# B&R Automation Studio project TD52 (part 72)

#### rtwtypes.h
```c
/********************************************************************
 * COPYRIGHT -- Bernecker + Rainer Industrie-Elektronik Ges.m.b.H.
 ********************************************************************
 * Program: LamStart
 * File: rtwtypes.h
 * Author: 105055527
 * Created: Thu May 18 17:26:11 2017
 ********************************************************************
 * Header for program LamStart
 ********************************************************************
 * Generated with B&R Automation Studio Target for Simulink V4.2
 * (ERT based)
 ********************************************************************/

#ifndef __RTWTYPES_H__
#define __RTWTYPES_H__
#ifndef TRUE
# define TRUE                          (1U)
#endif

#ifndef FALSE
# define FALSE                         (0U)
#endif

#ifndef __TMWTYPES__
#define __TMWTYPES__
#include <limits.h>

/*=======================================================================*
 * Target hardware information
 *   Device type: Intel->x86/Pentium
 *   Number of bits:     char:   8    short:   16    long:  32
 *                       long:  32
 *                       native word size:  32
 *   Byte ordering: LittleEndian
 *   Signed integer division rounds to: Zero
 *   Shift right on a signed integer as arithmetic shift: on
 *=======================================================================*/

/*=======================================================================*
 * Fixed width word size data types:                                     *
 *   int8_T, int16_T, int32_T     - signed 8, 16, or 32 bit integers     *
 *   uint8_T, uint16_T, uint32_T  - unsigned 8, 16, or 32 bit integers   *
 *   real32_T, real64_T           - 32 and 64 bit floating point numbers *
 *=======================================================================*/
typedef signed char int8_T;
typedef unsigned char uint8_T;
typedef short int16_T;
typedef unsigned short uint16_T;
typedef long int32_T;
typedef unsigned long uint32_T;
typedef float real32_T;
typedef double real64_T;

/*===========================================================================*
 * Generic type definitions: real_T, time_T, boolean_T, int_T, uint_T,       *
 *                           ulong_T, char_T and byte_T.                     *
 *===========================================================================*/
typedef double real_T;
typedef double time_T;
typedef unsigned char boolean_T;
typedef long int_T;
typedef unsigned long uint_T;
typedef unsigned long ulong_T;
typedef char char_T;
typedef unsigned char uchar_T;
typedef char_T byte_T;

/*=======================================================================*
 * Min and Max:                                                          *
 *   int8_T, int16_T, int32_T     - signed 8, 16, or 32 bit integers     *
 *   uint8_T, uint16_T, uint32_T  - unsigned 8, 16, or 32 bit integers   *
 *=======================================================================*/
#define MAX_int8_T                     ((int8_T)(127))
#define MIN_int8_T                     ((int8_T)(-128))
#define MAX_uint8_T                    ((uint8_T)(255U))
#define MIN_uint8_T                    ((uint8_T)(0U))
#define MAX_int16_T                    ((int16_T)(32767))
#define MIN_int16_T                    ((int16_T)(-32768))
#define MAX_uint16_T                   ((uint16_T)(65535U))
#define MIN_uint16_T                   ((uint16_T)(0U))
#define MAX_int32_T                    ((int32_T)(2147483647))
#define MIN_int32_T                    ((int32_T)(-2147483647-1))
#define MAX_uint32_T                   ((uint32_T)(0xFFFFFFFFU))
#define MIN_uint32_T                   ((uint32_T)(0U))

/* Logical type definitions */
#if (!defined(__cplusplus)) && (!defined(__true_false_are_keywords))
#  ifndef false
#   define false                       (0U)
#  endif

#  ifndef true
#   define true                        (1U)
#  endif
#endif

/*
 * Simulink Coder assumes the code is compiled on a target using a 2's complement representation
 * for signed integer values.
 */
#if ((SCHAR_MIN + 1) != -SCHAR_MAX)
#error "This code must be compiled using a 2's complement representation for signed integer values"
#endif

/* This ID is used to detect inclusion of an incompatible rtwtypes.h */
#define RTWTYPES_ID_C08S16I32L32N32F1
#else                                  /* __TMWTYPES__ */
#define TMWTYPES_PREVIOUSLY_INCLUDED
#endif                                 /* __TMWTYPES__ */

/* Block D-Work pointer type */
typedef void * pointer_T;

/* Simulink specific types */
#ifndef __SIMSTRUC_TYPES_H__
#define __SIMSTRUC_TYPES_H__

/* Trigger directions: falling, either, and rising */
typedef enum {
  FALLING_ZERO_CROSSING = -1,
  ANY_ZERO_CROSSING = 0,
  RISING_ZERO_CROSSING = 1
} ZCDirection;

/* Previous state of a trigger signal */
typedef uint8_T ZCSigState;

/* Initial value of a trigger zero crossing signal */
#define UNINITIALIZED_ZCSIG            0x03U
#define NEG_ZCSIG                      0x02U
#define POS_ZCSIG                      0x01U
#define ZERO_ZCSIG                     0x00U

/* Current state of a trigger signal */
typedef enum {
  FALLING_ZCEVENT = -1,
  NO_ZCEVENT = 0,
  RISING_ZCEVENT = 1
} ZCEventType;

#endif                                 /* __SIMSTRUC_TYPES_H__ */
#endif                                 /* __RTWTYPES_H__ */

#ifndef MIN
#define MIN(a,b)                       ((a) < (b) ? (a) : (b))
#endif

#ifndef MAX
#define MAX(a,b)                       ((a) > (b) ? (a) : (b))
#endif
```

#### LamStart.c
```c
/********************************************************************
 * COPYRIGHT -- Bernecker + Rainer Industrie-Elektronik Ges.m.b.H.
 ********************************************************************
 * Program: LamStart
 * File: LamStart.c
 * Author: 105055527
 * Created: Thu May 18 17:26:11 2017
 ********************************************************************
 * Implementation of program LamStart
 ********************************************************************
 * Generated with B&R Automation Studio Target for Simulink V4.2
 * (ERT based)
 ********************************************************************/
#include "LamStart.h"
#include "LamStart_private.h"

/*  Defines */
#define LamStart_POS_ZCSIG             ((uint8_T)1U)
#define LamStart_UNINITIALIZED_ZCSIG   ((uint8_T)3U)

/*  Data Types */

/**************************** GLOBAL DATA *************************************/
/*  Definitions */

/*  Declarations  */

/***************************** FILE SCOPE DATA ********************************/

/*************************** FUNCTIONS ****************************************/

/* Lookup Binary Search Utility BINARYSEARCH_real32_T */
void BINARYSEARCH_real32_T(uint32_T *piLeft, uint32_T *piRght, real32_T u, const
  real32_T *pData, uint32_T iHi, struct fLamStart* inst)
{
  /* Find the location of current input value in the data table. */
  *piLeft = 0U;
  *piRght = iHi;
  if (u <= pData[0] ) {
    /* Less than or equal to the smallest point in the table. */
    *piRght = 0U;
  } else if (u >= pData[iHi] ) {
    /* Greater than or equal to the largest point in the table. */
    *piLeft = iHi;
  } else {
    uint32_T i;

    /* Do a binary search. */
    while (( *piRght - *piLeft ) > 1U ) {
      /* Get the average of the left and right indices using to Floor rounding. */
      i = (*piLeft + *piRght) >> 1;

      /* Move either the right index or the left index so that */
      /*  LeftDataPoint <= CurrentValue < RightDataPoint */
      if (u < pData[i] ) {
        *piRght = i;
      } else {
        *piLeft = i;
      }
    }
  }
}

/* Lookup Utility LookUp_real32_T_real32_T */
void LookUp_real32_T_real32_T(real32_T *pY, const real32_T *pYData, real32_T u,
  const real32_T *pUData, uint32_T iHi, struct fLamStart* inst)
{
  uint32_T iLeft;
  uint32_T iRght;
  BINARYSEARCH_real32_T( &(iLeft), &(iRght), u, pUData, iHi, inst);

  {
    real32_T lambda;
    if (pUData[iRght] > pUData[iLeft] ) {
      real32_T num;
      real32_T den;
      den = pUData[iRght];
      den = den - pUData[iLeft];
      num = u;
      num = num - pUData[iLeft];
      lambda = num / den;
    } else {
      lambda = 0.0F;
    }

    {
      real32_T yLeftCast;
      real32_T yRghtCast;
      yLeftCast = pYData[iLeft];
      yRghtCast = pYData[iRght];
      yLeftCast += lambda * ( yRghtCast - yLeftCast );
      (*pY) = yLeftCast;
    }
  }
}

/* Model step function */
void LamStart_step(struct BlockIO_LamStart *LamStart_B, struct D_Work_LamStart *LamStart_DWork,
                   struct PrevZCSigStates_LamStart *LamStart_PrevZCSigState,
                   ExternalOutputs_LamStart *LamStart_Y, struct fLamStart* inst)
{
  /* local block i/o variables */
  real32_T rtb_LookupTableDynamic;
  real32_T rtb_TmpSignalConversionAtLookup[2];
  real32_T rtb_TmpSignalConversionAtLook_b[2];
  real32_T rtb_rLowerOilTemp;
  real32_T rtb_rLamLoLim_N_y[3];
  real32_T rtb_rLamLoLim_N_x[3];
  real32_T rtb_rN_Eng_h;
  real32_T rtb_LookupTableDynamic1;
  real32_T rtb_rT_EO;
  boolean_T rtb_LogicalOperator2;
  boolean_T didZcEventOccur;
  real32_T rtb_rHigherOilTemp;
  real32_T rtb_Abs1;
  real32_T rtb_Product;
  real32_T rtb_UkYk1;
  boolean_T rtb_Switch1;
  boolean_T rtb_RelationalOperator;

  /* S-Function (bur_bus_in): '<Root>/Bus Input2' */
  LamStart_B->BusInput2 = inst->Perm;

  /* Abs: '<S6>/Abs1' incorporates:
   *  BusSelector: '<S6>/Bus Selector7'
   */
  rtb_Abs1 = (real32_T)fabs(LamStart_B->BusInput2.rLamSlewRate);

  /* Product: '<S9>/delta rise limit' incorporates:
   *  SampleTimeMath: '<S9>/sample time'
   *
   * About '<S9>/sample time':
   *  y = K where K = ( w * Ts )
   */
  rtb_rHigherOilTemp = rtb_Abs1 * 0.01F;

  /* S-Function (bur_bus_in): '<Root>/Bus Input1' */
  LamStart_B->BusInput1 = inst->Para;

  /* S-Function (bur_bus_in): '<Root>/Bus Input' */
  LamStart_B->BusInput = inst->IN;

  /* BusSelector: '<Root>/Bus Selector3' */
  rtb_rLowerOilTemp = LamStart_B->BusInput.rN_Eng;

  /* BusSelector: '<Root>/Bus Selector13' */
  rtb_rLamLoLim_N_y[0] = LamStart_B->BusInput2.refPoint_Lam_N_Offs_x[0];
  rtb_rLamLoLim_N_y[1] = LamStart_B->BusInput2.refPoint_Lam_N_Offs_x[1];
  rtb_rLamLoLim_N_y[2] = LamStart_B->BusInput2.refPoint_Lam_N_Offs_x[2];
  rtb_rLamLoLim_N_x[0] = LamStart_B->BusInput2.refPoint_Lam_N_Offs_y[0];
  rtb_rLamLoLim_N_x[1] = LamStart_B->BusInput2.refPoint_Lam_N_Offs_y[1];
  rtb_rLamLoLim_N_x[2] = LamStart_B->BusInput2.refPoint_Lam_N_Offs_y[2];

  /* Dynamic Look-Up Table Block: '<Root>/Lookup Table Dynamic2'
   * Input0  Data Type:  Floating Point real32_T
   * Input1  Data Type:  Floating Point real32_T
   * Input2  Data Type:  Floating Point real32_T
   * Output0 Data Type:  Floating Point real32_T
   * Lookup Method: Linear_Endpoint
   *
   */
  LookUp_real32_T_real32_T( &(rtb_rT_EO), rtb_rLamLoLim_N_x, rtb_rLowerOilTemp,
    rtb_rLamLoLim_N_y, 2U, inst);

  /* Product: '<Root>/Product' */
  rtb_Product = LamStart_B->BusInput1.rLam_Start_Offs * rtb_rT_EO;

  /* Switch: '<S7>/Switch3' incorporates:
   *  Constant: '<S6>/Constant2'
   *  Constant: '<S6>/Constant4'
   *  Gain: '<S6>/Gain1'
   *  RelationalOperator: '<S7>/groesser '
   *  RelationalOperator: '<S7>/kleiner'
   *  Switch: '<S7>/Switch1'
   *  Switch: '<S7>/Switch2'
   *  UnitDelay: '<S7>/Unit Delay2'
   */
  if (LamStart_B->BusInput.bReset) {
    rtb_Switch1 = FALSE;
  } else if (LamStart_B->BusInput.rN_Eng < 10.0F) {
    /* Switch: '<S7>/Switch1' incorporates:
     *  Constant: '<S7>/FALSE'
     */
    rtb_Switch1 = FALSE;
  } else if (LamStart_B->BusInput.rN_Eng > 0.995F *
             LamStart_B->BusInput1.rN_EngNom) {
    /* Switch: '<S7>/Switch2' incorporates:
     *  Constant: '<S7>/TRUE'
     *  Switch: '<S7>/Switch1'
     */
    rtb_Switch1 = TRUE;
  } else {
    rtb_Switch1 = LamStart_DWork->UnitDelay2_DSTATE;
  }

  /* End of Switch: '<S7>/Switch3' */

  /* Outputs for Atomic SubSystem: '<S6>/TON' */
  /* Logic: '<S8>/Logical Operator2' */
  rtb_LogicalOperator2 = !rtb_Switch1;

  /* DiscreteIntegrator: '<S8>/Discrete-Time Integrator' */
  if (rtb_LogicalOperator2 || (LamStart_DWork->DiscreteTimeIntegrator_PrevRese
       != 0)) {
    LamStart_DWork->DiscreteTimeIntegrator_DSTATE = 0.0F;
  }

  /* RelationalOperator: '<S8>/Relational Operator' incorporates:
   *  DiscreteIntegrator: '<S8>/Discrete-Time Integrator'
   */
  rtb_RelationalOperator = (LamStart_DWork->DiscreteTimeIntegrator_DSTATE >=
    LamStart_B->BusInput2.rTi_idle);

  /* Update for DiscreteIntegrator: '<S8>/Discrete-Time Integrator' incorporates:
   *  DataTypeConversion: '<S10>/Conversion'
   *  Logic: '<S8>/Logical Operator'
   *  Logic: '<S8>/Logical Operator1'
   */
  LamStart_DWork->DiscreteTimeIntegrator_DSTATE += (real32_T)
    ((!rtb_RelationalOperator) && rtb_Switch1) * 0.01F;
  if (rtb_LogicalOperator2) {
    LamStart_DWork->DiscreteTimeIntegrator_PrevRese = 1;
  } else {
    LamStart_DWork->DiscreteTimeIntegrator_PrevRese = 0;
  }

  /* End of Update for DiscreteIntegrator: '<S8>/Discrete-Time Integrator' */

  /* Logic: '<S6>/Logical Operator' incorporates:
   *  Logic: '<S6>/Logical Operator1'
   *  Logic: '<S8>/Logical Operator3'
   */
  rtb_RelationalOperator = !((rtb_RelationalOperator && rtb_Switch1) ||
    LamStart_B->BusInput.bGCB_ON);

  /* End of Outputs for SubSystem: '<S6>/TON' */

  /* Delay: '<S9>/Delay' */
  didZcEventOccur = (((LamStart_PrevZCSigState->Delay_Reset_ZCE ==
                       LamStart_POS_ZCSIG) != rtb_RelationalOperator) &&
                     (LamStart_PrevZCSigState->Delay_Reset_ZCE !=
                      LamStart_UNINITIALIZED_ZCSIG));
  LamStart_PrevZCSigState->Delay_Reset_ZCE = (uint8_T)rtb_RelationalOperator;
  if (rtb_RelationalOperator || didZcEventOccur) {
    LamStart_DWork->icLoad = 1U;
  }

  if (LamStart_DWork->icLoad != 0) {
    LamStart_DWork->Delay_DSTATE = rtb_Product;
  }

  rtb_rT_EO = LamStart_DWork->Delay_DSTATE;

  /* End of Delay: '<S9>/Delay' */

  /* Switch: '<S9>/etaVolConst' incorporates:
   *  Constant: '<S6>/Constant6'
   */
  if (rtb_RelationalOperator) {
    rtb_UkYk1 = rtb_Product;
  } else {
    rtb_UkYk1 = 0.0F;
  }

  /* End of Switch: '<S9>/etaVolConst' */

  /* Sum: '<S9>/Difference Inputs1' */
  rtb_UkYk1 -= rtb_rT_EO;

  /* Switch: '<S11>/Switch2' incorporates:
   *  RelationalOperator: '<S11>/LowerRelop1'
   */
  if (!(rtb_UkYk1 > rtb_rHigherOilTemp)) {
    /* Product: '<S9>/delta fall limit' incorporates:
     *  Gain: '<S6>/Gain'
     */
    rtb_Abs1 = -rtb_Abs1 * 0.01F;

    /* Switch: '<S11>/Switch' incorporates:
     *  RelationalOperator: '<S11>/UpperRelop'
     */
    if (rtb_UkYk1 < rtb_Abs1) {
      rtb_rHigherOilTemp = rtb_Abs1;
    } else {
      rtb_rHigherOilTemp = rtb_UkYk1;
    }

    /* End of Switch: '<S11>/Switch' */
  }

  /* End of Switch: '<S11>/Switch2' */

  /* Sum: '<S9>/Difference Inputs2' */
  rtb_Abs1 = rtb_rHigherOilTemp + rtb_rT_EO;

  /* BusSelector: '<Root>/Bus Selector11' */
  rtb_rT_EO = LamStart_B->BusInput.rT_EO;

  /* BusSelector: '<Root>/Bus Selector10' */
  rtb_rLowerOilTemp = LamStart_B->BusInput2.rLowerOilTemp;
  rtb_rN_Eng_h = LamStart_B->BusInput2.rLowerOilLambda;
  rtb_LookupTableDynamic1 = LamStart_B->BusInput2.rHigherOilLambda;

  /* SignalConversion: '<Root>/TmpSignal ConversionAtLookup Table Dynamic1Inport2' incorporates:
   *  BusSelector: '<Root>/Bus Selector10'
   */
  rtb_TmpSignalConversionAtLookup[0] = rtb_rLowerOilTemp;
  rtb_TmpSignalConversionAtLookup[1] = LamStart_B->BusInput2.rHigherOilTemp;

  /* SignalConversion: '<Root>/TmpSignal ConversionAtLookup Table Dynamic1Inport3' */
  rtb_TmpSignalConversionAtLook_b[0] = rtb_rN_Eng_h;
  rtb_TmpSignalConversionAtLook_b[1] = rtb_LookupTableDynamic1;

  /* Dynamic Look-Up Table Block: '<Root>/Lookup Table Dynamic1'
   * Input0  Data Type:  Floating Point real32_T
   * Input1  Data Type:  Floating Point real32_T
   * Input2  Data Type:  Floating Point real32_T
   * Output0 Data Type:  Floating Point real32_T
   * Lookup Method: Linear_Endpoint
   *
   */
  LookUp_real32_T_real32_T( &(rtb_LookupTableDynamic1),
    rtb_TmpSignalConversionAtLook_b, rtb_rT_EO, rtb_TmpSignalConversionAtLookup,
    1U, inst);

  /* Sum: '<Root>/Add' */
  rtb_UkYk1 = rtb_LookupTableDynamic1 - rtb_Abs1;

  /* BusSelector: '<Root>/Bus Selector5' */
  rtb_rN_Eng_h = LamStart_B->BusInput.rN_Eng;

  /* BusSelector: '<Root>/Bus Selector8' */
  rtb_rLamLoLim_N_x[0] = LamStart_B->BusInput2.rLamLoLim_N_x[0];
  rtb_rLamLoLim_N_x[1] = LamStart_B->BusInput2.rLamLoLim_N_x[1];
  rtb_rLamLoLim_N_x[2] = LamStart_B->BusInput2.rLamLoLim_N_x[2];
  rtb_rLamLoLim_N_y[0] = LamStart_B->BusInput2.rLamLoLim_N_y[0];
  rtb_rLamLoLim_N_y[1] = LamStart_B->BusInput2.rLamLoLim_N_y[1];
  rtb_rLamLoLim_N_y[2] = LamStart_B->BusInput2.rLamLoLim_N_y[2];

  /* Dynamic Look-Up Table Block: '<Root>/Lookup Table Dynamic'
   * Input0  Data Type:  Floating Point real32_T
   * Input1  Data Type:  Floating Point real32_T
   * Input2  Data Type:  Floating Point real32_T
   * Output0 Data Type:  Floating Point real32_T
   * Lookup Method: Linear_Endpoint
   *
   */
  LookUp_real32_T_real32_T( &(rtb_LookupTableDynamic), rtb_rLamLoLim_N_y,
    rtb_rN_Eng_h, rtb_rLamLoLim_N_x, 2U, inst);

  /* Switch: '<S5>/Switch2' incorporates:
   *  Constant: '<Root>/Constant5'
   *  RelationalOperator: '<S5>/LowerRelop1'
   *  RelationalOperator: '<S5>/UpperRelop'
   *  Switch: '<S5>/Switch'
   */
  if (rtb_UkYk1 > 3.0F) {
    /* Outport: '<Root>/rLambda_start_idle' */
    LamStart_Y->rLambda_start_idle = 3.0F;
  } else if (rtb_UkYk1 < rtb_LookupTableDynamic) {
    /* Switch: '<S5>/Switch' incorporates:
     *  Outport: '<Root>/rLambda_start_idle'
     */
    LamStart_Y->rLambda_start_idle = rtb_LookupTableDynamic;
  } else {
    /* Outport: '<Root>/rLambda_start_idle' incorporates:
     *  Switch: '<S5>/Switch'
     */
    LamStart_Y->rLambda_start_idle = rtb_UkYk1;
  }

  /* End of Switch: '<S5>/Switch2' */

  /* Outport: '<Root>/dbg' incorporates:
   *  BusCreator: '<Root>/BusConversion_InsertedFor_dbg_at_inport_0'
   */
  LamStart_Y->dbg.rLambda_start = rtb_Abs1;
  LamStart_Y->dbg.rLambda_idle = rtb_LookupTableDynamic1;
  LamStart_Y->dbg.rLambda_start_raw = rtb_Product;
  LamStart_Y->dbg.rLamLim = rtb_LookupTableDynamic;

  /* BusCreator: '<Root>/BusConversion_InsertedFor_Bus Output1_at_inport_0' */
  LamStart_B->BusConversion_InsertedFor_BusOu.rLambda_start = rtb_Abs1;
  LamStart_B->BusConversion_InsertedFor_BusOu.rLambda_idle =
    rtb_LookupTableDynamic1;
  LamStart_B->BusConversion_InsertedFor_BusOu.rLambda_start_raw = rtb_Product;
  LamStart_B->BusConversion_InsertedFor_BusOu.rLamLim = rtb_LookupTableDynamic;

  /* S-Function (bur_bus_out): '<Root>/Bus Output1' */
  inst->dbg = LamStart_B->BusConversion_InsertedFor_BusOu;

  /* S-Function (bur_out): '<Root>/Output1' */
  inst->rLambda_start_idle = LamStart_Y->rLambda_start_idle;

  /* UnitDelay: '<S4>/Unit Delay' */
  LamStart_B->UnitDelay = LamStart_DWork->UnitDelay_DSTATE;

  /* S-Function (bur_out): '<Root>/Output' */
  inst->Version = LamStart_B->UnitDelay;

  /* Update for UnitDelay: '<S7>/Unit Delay2' */
  LamStart_DWork->UnitDelay2_DSTATE = rtb_Switch1;

  /* Update for Delay: '<S9>/Delay' */
  LamStart_DWork->icLoad = 0U;
  LamStart_DWork->Delay_DSTATE = rtb_Abs1;

  /* Update for UnitDelay: '<S4>/Unit Delay' */
  LamStart_DWork->UnitDelay_DSTATE = 1000U;
}

/* Model initialize function */
void LamStart_initialize(struct D_Work_LamStart *LamStart_DWork,
  struct PrevZCSigStates_LamStart *LamStart_PrevZCSigState, struct fLamStart* inst)
{
  LamStart_PrevZCSigState->Delay_Reset_ZCE = UNINITIALIZED_ZCSIG;

  /* InitializeConditions for Delay: '<S9>/Delay' */
  LamStart_DWork->icLoad = 1U;
}

/* Model terminate function */
void LamStart_terminate(struct fLamStart* inst)
{
  /* (no terminate code required) */
}

/*======================== TOOL VERSION INFORMATION ==========================*
 * MATLAB 8.0 (R2012b)20-Jul-2012                                             *
 * Simulink 8.0 (R2012b)20-Jul-2012                                           *
 * Simulink Coder 8.3 (R2012b)20-Jul-2012                                     *
 * Embedded Coder 6.3 (R2012b)20-Jul-2012                                     *
 * Stateflow 8.0 (R2012b)20-Jul-2012                                          *
 *============================================================================*/

/*======================= LICENSE IN USE INFORMATION =========================*
 * matlab                                                                     *
 * matlab_coder                                                               *
 * real-time_workshop                                                         *
 * rtw_embedded_coder                                                         *
 * simulink                                                                   *
 *============================================================================*/
```

#### fLamStart.c
```c
/********************************************************************
 * COPYRIGHT -- Bernecker + Rainer Industrie-Elektronik Ges.m.b.H.
 ********************************************************************
 * Program: LamStart
 * File: fLamStart.c
 * Author: 105055527
 * Created: Thu May 18 17:26:11 2017
 ********************************************************************
 * Implementation of program LamStart
 ********************************************************************
 * Generated with B&R Automation Studio Target for Simulink V4.2
 * (ERT based)
 ********************************************************************/
#include <bur/plctypes.h>
#include "LamStart.h"
#include "rtwtypes.h"

/* Defines */
#define SS_TERMINATE 4
#define SS_OUTPUT 3
#define SS_INITIALIZE 2

/*  Data Types */

/**************************** GLOBAL DATA *************************************/
/*  Definitions */

/*  Declarations  */

/***************************** FILE SCOPE DATA ********************************/

/*************************** FUNCTIONS ****************************************/
#ifdef __cplusplus

unsigned long bur_heap_size = 6553500;

#endif

void fLamStart(struct fLamStart* inst)
{
  BlockIO_LamStart *LamStart_B = &(inst)->bur_BlockIO_LamStart;
	D_Work_LamStart *LamStart_DWork = &(inst)->bur_D_Work_LamStart;
	PrevZCSigStates_LamStart *LamStart_PrevZCSigState = &(inst)->bur_PrevZCSigStates_LamStart;
	ExternalOutputs_LamStart *LamStart_Y = &(inst)->bur_ExternalOutputs_LamStart;

  switch (inst->ssMethodType)
  {
   case SS_INITIALIZE:
    /* call model initialize function */
    LamStart_initialize(LamStart_DWork, LamStart_PrevZCSigState, inst);
    break;

   case SS_OUTPUT:
    /* call model step function */
    LamStart_step(LamStart_B, LamStart_DWork, LamStart_PrevZCSigState,
                  LamStart_Y, inst);

    break;

   case SS_TERMINATE:
    /* call model terminate function */
    LamStart_terminate(inst);
    break;
  }
}

/*****************************************************************************
   Function block sample time: 0.01s
 *****************************************************************************/

/*****************************************************************************
   B&R Automation Studio Target for Simulink Version: A4.5.1 (27-Jul-2015)
 *****************************************************************************/

/*======================== TOOL VERSION INFORMATION ==========================*
 * MATLAB 8.0 (R2012b)20-Jul-2012                                             *
 * Simulink 8.0 (R2012b)20-Jul-2012                                           *
 * Simulink Coder 8.3 (R2012b)20-Jul-2012                                     *
 * Embedded Coder 6.3 (R2012b)20-Jul-2012                                     *
 * Stateflow 8.0 (R2012b)20-Jul-2012                                          *
 *============================================================================*/

/*======================= LICENSE IN USE INFORMATION =========================*
 * matlab                                                                     *
 * matlab_coder                                                               *
 * real-time_workshop                                                         *
 * rtw_embedded_coder                                                         *
 * simulink                                                                   *
 *============================================================================*/
```

#### lib_properties.txt
```
For manual assignment to hardware configuration please
add the following additional include directories:

\Logical\MATLAB_includes\R2012b\

And the following additional build options:

-lm -D MODEL=LamStart -D NUMST=1 -D NCSTATES=0 -D HAVESTDIO -D ONESTEPFCN=1 -D TERMFCN=1 -D MAT_FILE=0 -D MULTI_INSTANCE_CODE=1 -D INTEGER_CODE=0 -D MT=0 -D CLASSIC_INTERFACE=0 -D TID01EQ=0
```

### Library Logical/EngineController/Lib_EC/lCPP_Int (ANSIC)

#### lCPP_Int.fun
```iecst
FUNCTION_BLOCK fCPP_Int
  VAR_INPUT
    ssMethodType: SINT;
  END_VAR  VAR_INPUT
        In : tCPPI_IN; (**)
  END_VAR
  VAR_INPUT
        Para : tCPPI_PARA; (**)
  END_VAR
  VAR_INPUT
        Perm : tCPPI_PERM; (**)
  END_VAR
 VAR_OUTPUT
        Out : tCPPI_OUT; (**)
  END_VAR
 VAR_OUTPUT
        Dbg : tCPPI_DBUG; (**)
  END_VAR
  VAR_OUTPUT
        Version : UDINT; (**)
  END_VAR
	VAR
		bur_BlockIO_CPP_Int : BlockIO_CPP_Int;
	END_VAR
	VAR
		bur_D_Work_CPP_Int : D_Work_CPP_Int;
	END_VAR
	VAR
		bur_PrevZCSigStates_CPP_Int : PrevZCSigStates_CPP_Int;
	END_VAR
	VAR
		bur_ExternalOutputs_CPP_Int : ExternalOutputs_CPP_Int;
	END_VAR
END_FUNCTION_BLOCK
```

#### lCPP_Int.typ
```iecst
TYPE

   tCPPI_DBUG : STRUCT
        tiInt_NonEmpty : REAL; (*Integrator Non Empty elapsed time [s]*)
        rCPP_Err : REAL; (*Cylinder Peak Pressure Error [%]*)
        bECPG : BOOL; (*Engine Cycle Puls Generator*)
        bFCPG : BOOL; (*Filter Cycle Puls Generator*)
    END_STRUCT;

   tCPPI_IN : STRUCT
        bReset : BOOL; (*Reset CPP Integrator*)
        rPr_CPP : REAL; (*Cylinder Peak Pressure [bar]*)
        rN_Eng : REAL; (*Engine Actual Speed [1/min]*)
        bSensorErr : BOOL; (*Sensor Error active*)
        bLimpHomeExt : BOOL; (*Limp Home Extended Mode active*)
        tiSample : REAL; (*Function Block  Sampletime [s]*)
    END_STRUCT;

   tCPPI_OUT : STRUCT
        rPr_CPP_Filt : REAL; (*Cycle Peak Pressure filtered [bar]*)
        rPI_Dur_Offset : REAL; (*Port Injection Duration reduction offset [%]*)
        rCA_Ign_Offset : REAL; (*Ignition Point Timing reduction offset [°CA]*)
        rNum_CPP_Int : REAL; (*Integrator Level [%]*)
        bCPP_AbsLim : BOOL; (*Absolut Limit Integrator Level at 100%*)
        bCPP_AbsLim_LHE : BOOL; (*Absolut Limit Integrator Level at 100% for Extended Limp Home Mode*)
        bSkipCyl : BOOL; (*Skip Cylinder Ignition on Engine Shutdown*)
    END_STRUCT;

   tCPPI_PARA : STRUCT
        rPr_AbsLimHi : REAL; (*Peak Pressure Limit High High [bar]*)
        rPr_AbsLim : REAL; (*Peak Pressure Limit High [bar]*)
        rPr_AbsLimHi_LHE : REAL; (*Peak Pressure for Extended Limp Home Mode Limit High High [bar]*)
        rPr_AbsLim_LHE : REAL; (*Peak Pressure  for Extended Limp Home Mode Limit High [bar]*)
        rPI_Dur_Offset_Max : REAL; (*Port Injection Duration Reduction Offset maximum [%]*)
        rCA_Ign_Offset_Max : REAL; (*Ignition Point Timing Reduction Offset maximum [°CA]*)
    END_STRUCT;

   tCPPI_PERM : STRUCT
        rInt_Dec : REAL; (*Integrator Decent per Cycle Factor [%/Cycle]*)
        rInt_Power : REAL; (*Integrator Weighting Function Power Factor*)
        tiSensorFilter : REAL; (*Sensor Error Filtertime [s]*)
        tiInt_NonEmpty : REAL; (*Integrator Nonempty Time until Shutdown [s]*)
        rPI_Dur_IntLimLo : REAL; (*Integrator Level Limit for Port Injection Duration reduction Low [%]*)
        rPI_Dur_IntLimHi : REAL; (*Integrator Level Limit for Port Injection Duration reduction High [%]*)
        rIgn_IntLimLo : REAL; (*Integrator Level Limit for Ignition Point Timing reduction Low [%]*)
        rIgn_IntLimHi : REAL; (*Integrator Level Limit for Ignition Point Timing reduction High [%]*)
    END_STRUCT;
END_TYPE
TYPE
BlockIO_CPP_Int : STRUCT
	BusInput2 : tCPPI_PERM;
	BusInput : tCPPI_IN;
	BusInput1 : tCPPI_PARA;
	EnableOutput : REAL;
	EnableOutput_m : REAL;
	Saturadition : REAL;
	SensorErrorFilter : REAL;
	Divide3 : REAL;
	UnitDelay : UDINT;
END_STRUCT;
D_Work_CPP_Int : STRUCT
	DelayInput1_DSTATE : REAL;
	DiscreteTimeAccumulator_DSTATE : REAL;
	ResettableDelay_DSTATE : REAL;
	UnitDelay_DSTATE : UDINT;
	EngineCycleCounter_DSTATE : UINT;
	FilterCycleCounter_DSTATE : UINT;
	UnitDelay2_DSTATE : BOOL;
	UnitDelay1_DSTATE : BOOL;
	DelayInput1_DSTATE_c : BOOL;
	DelayInput1_DSTATE_f : BOOL;
	DiscreteTimeAccumulator_PrevRes : SINT;
END_STRUCT;
PrevZCSigStates_CPP_Int : STRUCT
	IgnitionPointandPIDurationOffse : USINT;
	CylinderPeakPressureIntegrator_ : USINT;
	ResettableDelay_Reset_ZCE : USINT;
	CylinderPeakPressureErrorCalcul : USINT;
END_STRUCT;
ExternalInputs_CPP_Int : STRUCT
	tCPPI_IN_o : tCPPI_IN;
	tCPPI_PARA_e : tCPPI_PARA;
	tCPPI_PERM_n : tCPPI_PERM;
END_STRUCT;
ExternalOutputs_CPP_Int : STRUCT
	tCPPI_OUT_c : tCPPI_OUT;
	tCPPI_DBUG_o : tCPPI_DBUG;
END_STRUCT;
END_TYPE
```

#### CPP_Int.h
```c
/********************************************************************
 * COPYRIGHT -- Bernecker + Rainer Industrie-Elektronik Ges.m.b.H.
 ********************************************************************
 * Program: CPP_Int
 * File: CPP_Int.h
 * Author: Messner
 * Created: Fri Nov 24 07:48:45 2017
 ********************************************************************
 * Header for program CPP_Int
 ********************************************************************
 * Generated with B&R Automation Studio Target for Simulink V4.2
 * (ERT based)
 ********************************************************************/

#ifndef RTW_HEADER_CPP_Int_h_
#define RTW_HEADER_CPP_Int_h_
#ifndef CPP_Int_COMMON_INCLUDES_
# define CPP_Int_COMMON_INCLUDES_
#include <math.h>
#include "rtwtypes.h"
#endif                                 /* CPP_Int_COMMON_INCLUDES_ */

#include "CPP_Int_types.h"
#include "lCPP_Int.h"

/* Macros for accessing real-time model data structure */
#ifndef rtmGetErrorStatus
# define rtmGetErrorStatus(rtm)        ((void*) 0)
#endif

#ifndef rtmSetErrorStatus
# define rtmSetErrorStatus(rtm, val)   ((void) 0)
#endif

#ifndef rtmGetStopRequested
# define rtmGetStopRequested(rtm)      ((void*) 0)
#endif

#ifndef MIN
#define MIN(a,b)                       ((a) < (b) ? (a) : (b))
#endif

#ifndef MAX
#define MAX(a,b)                       ((a) > (b) ? (a) : (b))
#endif

/* Block signals (auto storage) */

/* Block states (auto storage) for system '<Root>' */

/* Zero-crossing (trigger) state */

/* External inputs (root inport signals with auto storage) */

/* External outputs (root outports fed by signals with auto storage) */

/* Model entry point functions */
extern void CPP_Int_initialize(PrevZCSigStates_CPP_Int *CPP_Int_PrevZCSigState, struct fCPP_Int* inst);
extern void CPP_Int_step(BlockIO_CPP_Int *CPP_Int_B, D_Work_CPP_Int
  *CPP_Int_DWork, PrevZCSigStates_CPP_Int *CPP_Int_PrevZCSigState,
  ExternalOutputs_CPP_Int *CPP_Int_Y, struct fCPP_Int* inst);
extern void CPP_Int_terminate(struct fCPP_Int* inst);

/*-
 * The generated code includes comments that allow you to trace directly
 * back to the appropriate location in the model.  The basic format
 * is <system>/block_name, where system is the system number (uniquely
 * assigned by Simulink) and block_name is the name of the block.
 *
 * Use the MATLAB hilite_system command to trace the generated code back
 * to the model.  For example,
 *
 * hilite_system('<S3>')    - opens system 3
 * hilite_system('<S3>/Kp') - opens and selects block Kp which resides in S3
 *
 * Here is the system hierarchy for this model
 *
 * '<Root>' : 'CPP_Int'
 * '<S1>'   : 'CPP_Int/Cycle Phase Detector Clock'
 * '<S2>'   : 'CPP_Int/Cylinder Peak Pressure Error Calculator'
 * '<S3>'   : 'CPP_Int/Cylinder Peak Pressure Integrator'
 * '<S4>'   : 'CPP_Int/Detect Increase'
 * '<S5>'   : 'CPP_Int/Environment Controller'
 * '<S6>'   : 'CPP_Int/Environment Controller1'
 * '<S7>'   : 'CPP_Int/Environment Controller2'
 * '<S8>'   : 'CPP_Int/Ignition Point and PI Duration Offset Calculator'
 * '<S9>'   : 'CPP_Int/Info'
 * '<S10>'  : 'CPP_Int/Shutdown Procedures '
 * '<S11>'  : 'CPP_Int/Cycle Phase Detector Clock/Detect Increase'
 * '<S12>'  : 'CPP_Int/Cycle Phase Detector Clock/Divisor'
 * '<S13>'  : 'CPP_Int/Cycle Phase Detector Clock/Pressure Change Detect'
 * '<S14>'  : 'CPP_Int/Cycle Phase Detector Clock/RPM TO  SecPerCycle'
 * '<S15>'  : 'CPP_Int/Cycle Phase Detector Clock/Divisor/Data Type Conversion Inherited'
 * '<S16>'  : 'CPP_Int/Cylinder Peak Pressure Error Calculator/Divisor'
 * '<S17>'  : 'CPP_Int/Cylinder Peak Pressure Error Calculator/Saturation Dynamic'
 * '<S18>'  : 'CPP_Int/Cylinder Peak Pressure Error Calculator/Saturation Dynamic1'
 * '<S19>'  : 'CPP_Int/Cylinder Peak Pressure Error Calculator/Divisor/Data Type Conversion Inherited'
 * '<S20>'  : 'CPP_Int/Cylinder Peak Pressure Integrator/Compare To Zero'
 * '<S21>'  : 'CPP_Int/Cylinder Peak Pressure Integrator/Integrator'
 * '<S22>'  : 'CPP_Int/Ignition Point and PI Duration Offset Calculator/Ramp Limiter Ignition Point reduction'
 * '<S23>'  : 'CPP_Int/Ignition Point and PI Duration Offset Calculator/Ramp Limiter Port Injection Duration reduction'
 * '<S24>'  : 'CPP_Int/Ignition Point and PI Duration Offset Calculator/Ramp Limiter Ignition Point reduction/Lower Signal Limiter'
 * '<S25>'  : 'CPP_Int/Ignition Point and PI Duration Offset Calculator/Ramp Limiter Ignition Point reduction/Ramp Slope [k] - factor'
 * '<S26>'  : 'CPP_Int/Ignition Point and PI Duration Offset Calculator/Ramp Limiter Ignition Point reduction/Saturation Dynamic1'
 * '<S27>'  : 'CPP_Int/Ignition Point and PI Duration Offset Calculator/Ramp Limiter Ignition Point reduction/Signal Enabler'
 * '<S28>'  : 'CPP_Int/Ignition Point and PI Duration Offset Calculator/Ramp Limiter Ignition Point reduction/Upper Signal Limiter'
 * '<S29>'  : 'CPP_Int/Ignition Point and PI Duration Offset Calculator/Ramp Limiter Ignition Point reduction/Ramp Slope [k] - factor/Divisor'
 * '<S30>'  : 'CPP_Int/Ignition Point and PI Duration Offset Calculator/Ramp Limiter Ignition Point reduction/Ramp Slope [k] - factor/Divisor/Data Type Conversion Inherited'
 * '<S31>'  : 'CPP_Int/Ignition Point and PI Duration Offset Calculator/Ramp Limiter Port Injection Duration reduction/Lower Signal Limiter'
 * '<S32>'  : 'CPP_Int/Ignition Point and PI Duration Offset Calculator/Ramp Limiter Port Injection Duration reduction/Ramp Slope [k] - factor'
 * '<S33>'  : 'CPP_Int/Ignition Point and PI Duration Offset Calculator/Ramp Limiter Port Injection Duration reduction/Saturation Dynamic1'
 * '<S34>'  : 'CPP_Int/Ignition Point and PI Duration Offset Calculator/Ramp Limiter Port Injection Duration reduction/Signal Enabler'
 * '<S35>'  : 'CPP_Int/Ignition Point and PI Duration Offset Calculator/Ramp Limiter Port Injection Duration reduction/Upper Signal Limiter'
 * '<S36>'  : 'CPP_Int/Ignition Point and PI Duration Offset Calculator/Ramp Limiter Port Injection Duration reduction/Ramp Slope [k] - factor/Divisor'
 * '<S37>'  : 'CPP_Int/Ignition Point and PI Duration Offset Calculator/Ramp Limiter Port Injection Duration reduction/Ramp Slope [k] - factor/Divisor/Data Type Conversion Inherited'
 * '<S38>'  : 'CPP_Int/Shutdown Procedures /Integrator Nonempty'
 * '<S39>'  : 'CPP_Int/Shutdown Procedures /Integrator Full'
 * '<S40>'  : 'CPP_Int/Shutdown Procedures /TON Timer Integrator Nonempty'
 */
#endif                                 /* RTW_HEADER_CPP_Int_h_ */
```

#### CPP_Int_private.h
```c
/********************************************************************
 * COPYRIGHT -- Bernecker + Rainer Industrie-Elektronik Ges.m.b.H.
 ********************************************************************
 * Program: CPP_Int
 * File: CPP_Int_private.h
 * Author: Messner
 * Created: Fri Nov 24 07:48:45 2017
 ********************************************************************
 * Header for program CPP_Int
 ********************************************************************
 * Generated with B&R Automation Studio Target for Simulink V4.2
 * (ERT based)
 ********************************************************************/

#ifndef RTW_HEADER_CPP_Int_private_h_
#define RTW_HEADER_CPP_Int_private_h_
#include "rtwtypes.h"
#include <bur/plctypes.h>
#ifndef __RTWTYPES_H__
#error This file requires rtwtypes.h to be included
#else
#ifdef TMWTYPES_PREVIOUSLY_INCLUDED
#error This file requires rtwtypes.h to be included before tmwtypes.h
#else

/* Check for inclusion of an incorrect version of rtwtypes.h */
#ifndef RTWTYPES_ID_C08S16I32L32N32F1
#error This code was generated with a different "rtwtypes.h" than the file included
#endif                                 /* RTWTYPES_ID_C08S16I32L32N32F1 */
#endif                                 /* TMWTYPES_PREVIOUSLY_INCLUDED */
#endif                                 /* __RTWTYPES_H__ */

#ifndef MIN
#define MIN(a,b)                       ((a) < (b) ? (a) : (b))
#endif

#ifndef MAX
#define MAX(a,b)                       ((a) > (b) ? (a) : (b))
#endif

extern real32_T rt_roundf(real32_T u, struct fCPP_Int* inst);

/* Exported functions */
#endif                                 /* RTW_HEADER_CPP_Int_private_h_ */
```

#### CPP_Int_types.h
```c
/********************************************************************
 * COPYRIGHT -- Bernecker + Rainer Industrie-Elektronik Ges.m.b.H.
 ********************************************************************
 * Program: CPP_Int
 * File: CPP_Int_types.h
 * Author: Messner
 * Created: Fri Nov 24 07:48:45 2017
 ********************************************************************
 * Header for program CPP_Int
 ********************************************************************
 * Generated with B&R Automation Studio Target for Simulink V4.2
 * (ERT based)
 ********************************************************************/

#ifndef RTW_HEADER_CPP_Int_types_h_
#define RTW_HEADER_CPP_Int_types_h_
#include "rtwtypes.h"
#ifndef MIN
#define MIN(a,b)                       ((a) < (b) ? (a) : (b))
#endif

#ifndef MAX
#define MAX(a,b)                       ((a) > (b) ? (a) : (b))
#endif

#endif                                 /* RTW_HEADER_CPP_Int_types_h_ */
```

#### rtwtypes.h
```c
/********************************************************************
 * COPYRIGHT -- Bernecker + Rainer Industrie-Elektronik Ges.m.b.H.
 ********************************************************************
 * Program: CPP_Int
 * File: rtwtypes.h
 * Author: Messner
 * Created: Fri Nov 24 07:48:45 2017
 ********************************************************************
 * Header for program CPP_Int
 ********************************************************************
 * Generated with B&R Automation Studio Target for Simulink V4.2
 * (ERT based)
 ********************************************************************/

#ifndef __RTWTYPES_H__
#define __RTWTYPES_H__
#ifndef TRUE
# define TRUE                          (1U)
#endif

#ifndef FALSE
# define FALSE                         (0U)
#endif

#ifndef __TMWTYPES__
#define __TMWTYPES__
#include <limits.h>

/*=======================================================================*
 * Target hardware information
 *   Device type: Intel->x86/Pentium
 *   Number of bits:     char:   8    short:   16    long:  32
 *                       long:  32
 *                       native word size:  32
 *   Byte ordering: LittleEndian
 *   Signed integer division rounds to: Zero
 *   Shift right on a signed integer as arithmetic shift: on
 *=======================================================================*/

/*=======================================================================*
 * Fixed width word size data types:                                     *
 *   int8_T, int16_T, int32_T     - signed 8, 16, or 32 bit integers     *
 *   uint8_T, uint16_T, uint32_T  - unsigned 8, 16, or 32 bit integers   *
 *   real32_T, real64_T           - 32 and 64 bit floating point numbers *
 *=======================================================================*/
typedef signed char int8_T;
typedef unsigned char uint8_T;
typedef short int16_T;
typedef unsigned short uint16_T;
typedef long int32_T;
typedef unsigned long uint32_T;
typedef float real32_T;
typedef double real64_T;

/*===========================================================================*
 * Generic type definitions: real_T, time_T, boolean_T, int_T, uint_T,       *
 *                           ulong_T, char_T and byte_T.                     *
 *===========================================================================*/
typedef double real_T;
typedef double time_T;
typedef unsigned char boolean_T;
typedef long int_T;
typedef unsigned long uint_T;
typedef unsigned long ulong_T;
typedef char char_T;
typedef unsigned char uchar_T;
typedef char_T byte_T;

/*=======================================================================*
 * Min and Max:                                                          *
 *   int8_T, int16_T, int32_T     - signed 8, 16, or 32 bit integers     *
 *   uint8_T, uint16_T, uint32_T  - unsigned 8, 16, or 32 bit integers   *
 *=======================================================================*/
#define MAX_int8_T                     ((int8_T)(127))
#define MIN_int8_T                     ((int8_T)(-128))
#define MAX_uint8_T                    ((uint8_T)(255U))
#define MIN_uint8_T                    ((uint8_T)(0U))
#define MAX_int16_T                    ((int16_T)(32767))
#define MIN_int16_T                    ((int16_T)(-32768))
#define MAX_uint16_T                   ((uint16_T)(65535U))
#define MIN_uint16_T                   ((uint16_T)(0U))
#define MAX_int32_T                    ((int32_T)(2147483647))
#define MIN_int32_T                    ((int32_T)(-2147483647-1))
#define MAX_uint32_T                   ((uint32_T)(0xFFFFFFFFU))
#define MIN_uint32_T                   ((uint32_T)(0U))

/* Logical type definitions */
#if (!defined(__cplusplus)) && (!defined(__true_false_are_keywords))
#  ifndef false
#   define false                       (0U)
#  endif

#  ifndef true
#   define true                        (1U)
#  endif
#endif

/*
 * Simulink Coder assumes the code is compiled on a target using a 2's complement representation
 * for signed integer values.
 */
#if ((SCHAR_MIN + 1) != -SCHAR_MAX)
#error "This code must be compiled using a 2's complement representation for signed integer values"
#endif

/* This ID is used to detect inclusion of an incompatible rtwtypes.h */
#define RTWTYPES_ID_C08S16I32L32N32F1
#else                                  /* __TMWTYPES__ */
#define TMWTYPES_PREVIOUSLY_INCLUDED
#endif                                 /* __TMWTYPES__ */

/* Block D-Work pointer type */
typedef void * pointer_T;

/* Simulink specific types */
#ifndef __SIMSTRUC_TYPES_H__
#define __SIMSTRUC_TYPES_H__

/* Trigger directions: falling, either, and rising */
typedef enum {
  FALLING_ZERO_CROSSING = -1,
  ANY_ZERO_CROSSING = 0,
  RISING_ZERO_CROSSING = 1
} ZCDirection;

/* Previous state of a trigger signal */
typedef uint8_T ZCSigState;

/* Initial value of a trigger zero crossing signal */
#define UNINITIALIZED_ZCSIG            0x03U
#define NEG_ZCSIG                      0x02U
#define POS_ZCSIG                      0x01U
#define ZERO_ZCSIG                     0x00U

/* Current state of a trigger signal */
typedef enum {
  FALLING_ZCEVENT = -1,
  NO_ZCEVENT = 0,
  RISING_ZCEVENT = 1
} ZCEventType;

#endif                                 /* __SIMSTRUC_TYPES_H__ */
#endif                                 /* __RTWTYPES_H__ */

#ifndef MIN
#define MIN(a,b)                       ((a) < (b) ? (a) : (b))
#endif

#ifndef MAX
#define MAX(a,b)                       ((a) > (b) ? (a) : (b))
#endif
```

#### CPP_Int.c
```c
/********************************************************************
 * COPYRIGHT -- Bernecker + Rainer Industrie-Elektronik Ges.m.b.H.
 ********************************************************************
 * Program: CPP_Int
 * File: CPP_Int.c
 * Author: Messner
 * Created: Fri Nov 24 07:48:45 2017
 ********************************************************************
 * Implementation of program CPP_Int
 ********************************************************************
 * Generated with B&R Automation Studio Target for Simulink V4.2
 * (ERT based)
 ********************************************************************/
#include "CPP_Int.h"
#include "CPP_Int_private.h"

/*  Defines */
#define CPP_Int_POS_ZCSIG              ((uint8_T)1U)
#define CPP_Int_UNINITIALIZED_ZCSIG    ((uint8_T)3U)

/*  Data Types */

/**************************** GLOBAL DATA *************************************/
/*  Definitions */

/*  Declarations  */

/***************************** FILE SCOPE DATA ********************************/

/*************************** FUNCTIONS ****************************************/
real32_T rt_roundf(real32_T u, struct fCPP_Int* inst)
{
  real32_T y;
  if ((real32_T)fabs(u) < 8.388608E+6F) {
    if (u >= 0.5F) {
      y = (real32_T)floor(u + 0.5F);
    } else if (u > -0.5F) {
      y = 0.0F;
    } else {
      y = (real32_T)ceil(u - 0.5F);
    }
  } else {
    y = u;
  }

  return y;
}

/* Model step function */
void CPP_Int_step(struct BlockIO_CPP_Int *CPP_Int_B, struct D_Work_CPP_Int *CPP_Int_DWork,
                  struct PrevZCSigStates_CPP_Int *CPP_Int_PrevZCSigState,
                  ExternalOutputs_CPP_Int *CPP_Int_Y, struct fCPP_Int* inst)
{
  /* local block i/o variables */
  boolean_T rtb_Reset;
  real32_T rtb_Switch_j;
  uint16_T rtb_OneSamplebeforenextCycle;
  uint16_T rtb_Subtract3_h;
  boolean_T rtb_LogicalOperator3;
  boolean_T rtb_FixPtRelationalOperator_h;
  uint16_T rtb_Subtract1;
  boolean_T rtb_RelationalOperator1;
  boolean_T rtb_LogicalOperator2;
  boolean_T rtb_LogicalOperator1_j;
  real32_T rtb_rPr_AbsLimHi_k;
  real32_T rtb_Switch_g;
  boolean_T rtb_LimitReached;
  real32_T rtb_rPr_AbsLim_h;
  uint16_T u;

  /* S-Function (bur_bus_in): '<Root>/Bus Input' */
  CPP_Int_B->BusInput = inst->In;

  /* S-Function (bur_bus_in): '<Root>/Bus Input1' */
  CPP_Int_B->BusInput1 = inst->Para;

  /* Delay: '<S1>/Engine Cycle Counter' incorporates:
   *  UnitDelay: '<S1>/Unit Delay1'
   */
  if (CPP_Int_DWork->UnitDelay1_DSTATE) {
    CPP_Int_DWork->EngineCycleCounter_DSTATE = 0U;
  }

  /* Sum: '<S1>/Subtract3' incorporates:
   *  Delay: '<S1>/Engine Cycle Counter'
   */
  rtb_Subtract3_h = (uint16_T)((uint32_T)
    CPP_Int_DWork->EngineCycleCounter_DSTATE + 1U);

  /* Switch: '<S12>/Switch' incorporates:
   *  Abs: '<S12>/Abs'
   *  BusSelector: '<Root>/Bus Selector7'
   *  RelationalOperator: '<S12>/Relational Operator'
   */
  if (2.22044605E-16F >= (real32_T)fabs(CPP_Int_B->BusInput.tiSample)) {
    rtb_Switch_j = 2.22044605E-16F;
  } else {
    rtb_Switch_j = CPP_Int_B->BusInput.tiSample;
  }

  /* End of Switch: '<S12>/Switch' */

  /* MinMax: '<S14>/MinMax' incorporates:
   *  BusSelector: '<Root>/Bus Selector7'
   */
  if (CPP_Int_B->BusInput.rN_Eng >= 100.0F) {
    rtb_rPr_AbsLimHi_k = CPP_Int_B->BusInput.rN_Eng;
  } else {
    rtb_rPr_AbsLimHi_k = 100.0F;
  }

  /* Product: '<S1>/Samples  Per Cycle' incorporates:
   *  Constant: '<S14>/Constant2'
   *  MinMax: '<S14>/MinMax'
   *  Product: '<S14>/Divide'
   */
  rtb_rPr_AbsLimHi_k = (real32_T)fmod(rt_roundf(1.0F / rtb_rPr_AbsLimHi_k *
    120.0F / rtb_Switch_j, inst), 65536.0F);
  rtb_OneSamplebeforenextCycle = (uint16_T)(rtb_rPr_AbsLimHi_k < 0.0F ?
    (uint16_T)(int32_T)(int16_T)-(int16_T)(uint16_T)-rtb_rPr_AbsLimHi_k :
    (uint16_T)rtb_rPr_AbsLimHi_k);

  /* Logic: '<S1>/Logical Operator3' incorporates:
   *  RelationalOperator: '<S13>/FixPt Relational Operator'
   *  RelationalOperator: '<S1>/Relational Operator'
   *  UnitDelay: '<S13>/Delay Input1'
   */
  rtb_LogicalOperator3 = ((rtb_Subtract3_h >= rtb_OneSamplebeforenextCycle) ||
    (CPP_Int_B->BusInput.rPr_CPP != CPP_Int_DWork->DelayInput1_DSTATE));

  /* RelationalOperator: '<S11>/FixPt Relational Operator' incorporates:
   *  UnitDelay: '<S11>/Delay Input1'
   */
  rtb_FixPtRelationalOperator_h = ((int32_T)rtb_LogicalOperator3 > (int32_T)
    CPP_Int_DWork->DelayInput1_DSTATE_c);

  /* Delay: '<S1>/Filter Cycle Counter' incorporates:
   *  Logic: '<S1>/Logical Operator4'
   *  UnitDelay: '<S1>/Unit Delay2'
   */
  if (CPP_Int_DWork->UnitDelay2_DSTATE || rtb_FixPtRelationalOperator_h) {
    CPP_Int_DWork->FilterCycleCounter_DSTATE = 0U;
  }

  /* Sum: '<S1>/Subtract1' incorporates:
   *  Delay: '<S1>/Filter Cycle Counter'
   *  Logic: '<S1>/One Cycle Self-locking'
   */
  rtb_Subtract1 = (uint16_T)((uint32_T)
    ((CPP_Int_DWork->FilterCycleCounter_DSTATE != 0) ||
     rtb_FixPtRelationalOperator_h) + (uint32_T)
    CPP_Int_DWork->FilterCycleCounter_DSTATE);

  /* S-Function (bur_bus_in): '<Root>/Bus Input2' */
  CPP_Int_B->BusInput2 = inst->Perm;

  /* Sum: '<S1>/One Sample before next Cycle' incorporates:
   *  Constant: '<S1>/act2'
   */
  rtb_OneSamplebeforenextCycle--;

  /* Product: '<S1>/Samples Per Cycle' incorporates:
   *  BusSelector: '<Root>/Bus Selector6'
   */
  rtb_rPr_AbsLimHi_k = (real32_T)fmod(rt_roundf
    (CPP_Int_B->BusInput2.tiSensorFilter / rtb_Switch_j, inst), 65536.0F);

  /* MinMax: '<S1>/MinMax1' incorporates:
   *  Product: '<S1>/Samples Per Cycle'
   */
  u = (uint16_T)(rtb_rPr_AbsLimHi_k < 0.0F ? (uint16_T)(int32_T)(int16_T)
                 -(int16_T)(uint16_T)-rtb_rPr_AbsLimHi_k : (uint16_T)
                 rtb_rPr_AbsLimHi_k);
  if (u <= rtb_OneSamplebeforenextCycle) {
    rtb_OneSamplebeforenextCycle = u;
  }

  /* End of MinMax: '<S1>/MinMax1' */

  /* Saturate: '<S1>/Limit Cycle Count' */
  if (!(rtb_OneSamplebeforenextCycle <= 1000)) {
    rtb_OneSamplebeforenextCycle = 1000U;
  }

  /* RelationalOperator: '<S1>/Relational Operator1' incorporates:
   *  Saturate: '<S1>/Limit Cycle Count'
   */
  rtb_RelationalOperator1 = (rtb_Subtract1 > rtb_OneSamplebeforenextCycle);

  /* Logic: '<Root>/Logical Operator2' incorporates:
   *  RelationalOperator: '<S4>/FixPt Relational Operator'
   *  UnitDelay: '<S4>/Delay Input1'
   */
  rtb_LogicalOperator2 = (rtb_RelationalOperator1 || ((int32_T)
    CPP_Int_B->BusInput.bReset > (int32_T)CPP_Int_DWork->DelayInput1_DSTATE_f));

  /* Outputs for Triggered SubSystem: '<Root>/Cylinder Peak Pressure Error Calculator' incorporates:
   *  TriggerPort: '<S2>/Trigger'
   */
  if (rtb_LogicalOperator2 &&
      (CPP_Int_PrevZCSigState->CylinderPeakPressureErrorCalcul != POS_ZCSIG)) {
    /* Switch: '<S2>/Switch2' */
    if (CPP_Int_B->BusInput.bLimpHomeExt) {
      rtb_rPr_AbsLimHi_k = CPP_Int_B->BusInput1.rPr_AbsLimHi_LHE;
    } else {
      rtb_rPr_AbsLimHi_k = CPP_Int_B->BusInput1.rPr_AbsLimHi;
    }

    /* End of Switch: '<S2>/Switch2' */

    /* Switch: '<S2>/Switch1' */
    if (CPP_Int_B->BusInput.bLimpHomeExt) {
      rtb_rPr_AbsLim_h = CPP_Int_B->BusInput1.rPr_AbsLim_LHE;
    } else {
      rtb_rPr_AbsLim_h = CPP_Int_B->BusInput1.rPr_AbsLim;
    }

    /* End of Switch: '<S2>/Switch1' */

    /* Switch: '<S18>/Switch' incorporates:
     *  Constant: '<S2>/act2'
     *  RelationalOperator: '<S18>/LowerRelop1'
     *  RelationalOperator: '<S18>/UpperRelop'
     *  Sum: '<S2>/Subtract2'
     *  Switch: '<S18>/Switch2'
     */
    if ((!(rtb_rPr_AbsLimHi_k > rtb_rPr_AbsLimHi_k)) && (rtb_rPr_AbsLimHi_k <
         1.0F + rtb_rPr_AbsLim_h)) {
      rtb_rPr_AbsLimHi_k = 1.0F + rtb_rPr_AbsLim_h;
    }

    /* End of Switch: '<S18>/Switch' */

    /* Sum: '<S2>/Pressure Limit Deviation [bar]' */
    rtb_rPr_AbsLimHi_k -= rtb_rPr_AbsLim_h;

    /* Switch: '<S16>/Switch' incorporates:
     *  Abs: '<S16>/Abs'
     *  RelationalOperator: '<S16>/Relational Operator'
     */
    if (2.22044605E-16F >= (real32_T)fabs(rtb_rPr_AbsLimHi_k)) {
      rtb_Switch_g = 2.22044605E-16F;
    } else {
      rtb_Switch_g = rtb_rPr_AbsLimHi_k;
    }

    /* End of Switch: '<S16>/Switch' */

    /* Switch: '<S2>/Sensor Error Filter' incorporates:
     *  Gain: '<S2>/Gain'
     */
    if (CPP_Int_B->BusInput.bSensorErr) {
      CPP_Int_B->SensorErrorFilter = 0.75F * rtb_rPr_AbsLim_h;
    } else {
      CPP_Int_B->SensorErrorFilter = CPP_Int_B->BusInput.rPr_CPP;
    }

    /* End of Switch: '<S2>/Sensor Error Filter' */

    /* Sum: '<S2>/Pressure Error [bar]' */
    rtb_Switch_j = CPP_Int_B->SensorErrorFilter - rtb_rPr_AbsLim_h;

    /* Switch: '<S17>/Switch2' incorporates:
     *  RelationalOperator: '<S17>/LowerRelop1'
     */
    if (!(rtb_Switch_j > rtb_rPr_AbsLimHi_k)) {
      /* Switch: '<S17>/Switch' incorporates:
       *  Constant: '<S2>/act1'
       *  RelationalOperator: '<S17>/UpperRelop'
       */
      if (rtb_Switch_j < 0.0F) {
        rtb_rPr_AbsLimHi_k = 0.0F;
      } else {
        rtb_rPr_AbsLimHi_k = rtb_Switch_j;
      }

      /* End of Switch: '<S17>/Switch' */
    }

    /* End of Switch: '<S17>/Switch2' */

    /* Product: '<S2>/Divide3' incorporates:
     *  DataTypeConversion: '<S2>/Data Type Conversion'
     *  Logic: '<S2>/Logical Operator2'
     */
    CPP_Int_B->Divide3 = (real32_T)!CPP_Int_B->BusInput.bReset / rtb_Switch_g *
      rtb_rPr_AbsLimHi_k;
  }

  CPP_Int_PrevZCSigState->CylinderPeakPressureErrorCalcul = (uint8_T)
    (rtb_LogicalOperator2 ? (int32_T)POS_ZCSIG : (int32_T)ZERO_ZCSIG);

  /* End of Outputs for SubSystem: '<Root>/Cylinder Peak Pressure Error Calculator' */

  /* Outputs for Triggered SubSystem: '<Root>/Cylinder Peak Pressure Integrator' incorporates:
   *  TriggerPort: '<S3>/Trigger'
   */
  if (rtb_LogicalOperator2 &&
      (CPP_Int_PrevZCSigState->CylinderPeakPressureIntegrator_ != POS_ZCSIG)) {
    /* Delay: '<S21>/Resettable Delay' */
    rtb_LimitReached = (((CPP_Int_PrevZCSigState->ResettableDelay_Reset_ZCE ==
                          CPP_Int_POS_ZCSIG) != CPP_Int_B->BusInput.bReset) &&
                        (CPP_Int_PrevZCSigState->ResettableDelay_Reset_ZCE !=
                         CPP_Int_UNINITIALIZED_ZCSIG));
    CPP_Int_PrevZCSigState->ResettableDelay_Reset_ZCE = (uint8_T)
      CPP_Int_B->BusInput.bReset;
    if (CPP_Int_B->BusInput.bReset || rtb_LimitReached) {
      CPP_Int_DWork->ResettableDelay_DSTATE = 0.0F;
    }

    /* Switch: '<S3>/Switch4' incorporates:
     *  Constant: '<S20>/Constant'
     *  Gain: '<S3>/Decent'
     *  Math: '<S3>/Power Weighting Function'
     *  RelationalOperator: '<S20>/Compare'
     */
    if (CPP_Int_B->Divide3 <= 0.0F) {
      rtb_Switch_j = -CPP_Int_B->BusInput2.rInt_Dec;
    } else if ((CPP_Int_B->Divide3 < 0.0F) && (CPP_Int_B->BusInput2.rInt_Power >
                (real32_T)floor(CPP_Int_B->BusInput2.rInt_Power))) {
      /* Math: '<S3>/Power Weighting Function' */
      rtb_Switch_j = -(real32_T)pow(-CPP_Int_B->Divide3,
        CPP_Int_B->BusInput2.rInt_Power);
    } else {
      /* Math: '<S3>/Power Weighting Function' */
      rtb_Switch_j = (real32_T)pow(CPP_Int_B->Divide3,
        CPP_Int_B->BusInput2.rInt_Power);
    }

    /* End of Switch: '<S3>/Switch4' */

    /* Sum: '<S21>/Subtract3' incorporates:
     *  Delay: '<S21>/Resettable Delay'
     */
    rtb_rPr_AbsLimHi_k = CPP_Int_DWork->ResettableDelay_DSTATE + rtb_Switch_j;

    /* Saturate: '<S21>/Saturadition' */
    if (rtb_rPr_AbsLimHi_k >= 1.0F) {
      CPP_Int_B->Saturadition = 1.0F;
    } else if (rtb_rPr_AbsLimHi_k <= 0.0F) {
      CPP_Int_B->Saturadition = 0.0F;
    } else {
      CPP_Int_B->Saturadition = rtb_rPr_AbsLimHi_k;
    }

    /* End of Saturate: '<S21>/Saturadition' */

    /* Update for Delay: '<S21>/Resettable Delay' */
    CPP_Int_DWork->ResettableDelay_DSTATE = CPP_Int_B->Saturadition;
  }

  CPP_Int_PrevZCSigState->CylinderPeakPressureIntegrator_ = (uint8_T)
    (rtb_LogicalOperator2 ? (int32_T)POS_ZCSIG : (int32_T)ZERO_ZCSIG);

  /* End of Outputs for SubSystem: '<Root>/Cylinder Peak Pressure Integrator' */

  /* Outputs for Triggered SubSystem: '<Root>/Ignition Point and PI Duration Offset Calculator' incorporates:
   *  TriggerPort: '<S8>/Trigger'
   */
  if (rtb_LogicalOperator2 &&
      (CPP_Int_PrevZCSigState->IgnitionPointandPIDurationOffse != POS_ZCSIG)) {
    /* Switch: '<S24>/Switch2' incorporates:
     *  Constant: '<S22>/act2'
     *  RelationalOperator: '<S24>/LowerRelop1'
     *  RelationalOperator: '<S24>/UpperRelop'
     *  Switch: '<S24>/Switch'
     */
    if (CPP_Int_B->BusInput2.rIgn_IntLimLo > CPP_Int_B->BusInput2.rIgn_IntLimHi)
    {
      rtb_Switch_j = CPP_Int_B->BusInput2.rIgn_IntLimHi;
    } else if (CPP_Int_B->BusInput2.rIgn_IntLimLo < 0.0F) {
      /* Switch: '<S24>/Switch' incorporates:
       *  Constant: '<S22>/act2'
       */
      rtb_Switch_j = 0.0F;
    } else {
      rtb_Switch_j = CPP_Int_B->BusInput2.rIgn_IntLimLo;
    }

    /* End of Switch: '<S24>/Switch2' */

    /* RelationalOperator: '<S27>/Limit Reached' */
    rtb_LimitReached = (CPP_Int_B->Saturadition >= rtb_Switch_j);

    /* Switch: '<S28>/Switch2' incorporates:
     *  Constant: '<S22>/act3'
     *  RelationalOperator: '<S28>/LowerRelop1'
     *  RelationalOperator: '<S28>/UpperRelop'
     *  Switch: '<S28>/Switch'
     */
    if (CPP_Int_B->BusInput2.rIgn_IntLimHi > 1.0F) {
      rtb_rPr_AbsLimHi_k = 1.0F;
    } else if (CPP_Int_B->BusInput2.rIgn_IntLimHi <
               CPP_Int_B->BusInput2.rIgn_IntLimLo) {
      /* Switch: '<S28>/Switch' */
      rtb_rPr_AbsLimHi_k = CPP_Int_B->BusInput2.rIgn_IntLimLo;
    } else {
      rtb_rPr_AbsLimHi_k = CPP_Int_B->BusInput2.rIgn_IntLimHi;
    }

    /* End of Switch: '<S28>/Switch2' */

    /* Sum: '<S22>/Delta X' */
    rtb_rPr_AbsLim_h = rtb_rPr_AbsLimHi_k - rtb_Switch_j;

    /* Switch: '<S29>/Switch' incorporates:
     *  Abs: '<S29>/Abs'
     *  RelationalOperator: '<S29>/Relational Operator'
     */
    if (2.22044605E-16F >= (real32_T)fabs(rtb_rPr_AbsLim_h)) {
      rtb_rPr_AbsLim_h = 2.22044605E-16F;
    }

    /* End of Switch: '<S29>/Switch' */

    /* Product: '<S22>/y = k * (x - d)' incorporates:
     *  DataTypeConversion: '<S27>/Data Type Conversion'
     *  Gain: '<S8>/Ignition Point reduction'
     *  Product: '<S25>/[k] - factor'
     *  Product: '<S27>/Enable Signal'
     *  Sum: '<S22>/Level Offset [x - d]'
     */
    rtb_Switch_j = ((real32_T)rtb_LimitReached * CPP_Int_B->Saturadition -
                    rtb_Switch_j) * (1.0F / rtb_rPr_AbsLim_h *
      -CPP_Int_B->BusInput1.rCA_Ign_Offset_Max);

    /* Switch: '<S26>/Switch2' incorporates:
     *  Constant: '<S22>/act1'
     *  Gain: '<S8>/Ignition Point reduction'
     *  RelationalOperator: '<S26>/LowerRelop1'
     *  RelationalOperator: '<S26>/UpperRelop'
     *  Switch: '<S26>/Switch'
     */
    if (rtb_Switch_j > 0.0F) {
      rtb_Switch_j = 0.0F;
    } else {
      if (rtb_Switch_j < -CPP_Int_B->BusInput1.rCA_Ign_Offset_Max) {
        /* Switch: '<S26>/Switch' incorporates:
         *  Gain: '<S8>/Ignition Point reduction'
         */
        rtb_Switch_j = -CPP_Int_B->BusInput1.rCA_Ign_Offset_Max;
      }
    }

    /* End of Switch: '<S26>/Switch2' */

    /* Product: '<S22>/Enable Output' incorporates:
     *  DataTypeConversion: '<S22>/Data Type Conversion'
     */
    CPP_Int_B->EnableOutput = (real32_T)rtb_LimitReached * rtb_Switch_j;

    /* Switch: '<S31>/Switch2' incorporates:
     *  Constant: '<S23>/act2'
     *  RelationalOperator: '<S31>/LowerRelop1'
     *  RelationalOperator: '<S31>/UpperRelop'
     *  Switch: '<S31>/Switch'
     */
    if (CPP_Int_B->BusInput2.rPI_Dur_IntLimLo >
        CPP_Int_B->BusInput2.rPI_Dur_IntLimHi) {
      rtb_Switch_j = CPP_Int_B->BusInput2.rPI_Dur_IntLimHi;
    } else if (CPP_Int_B->BusInput2.rPI_Dur_IntLimLo < 0.0F) {
      /* Switch: '<S31>/Switch' incorporates:
       *  Constant: '<S23>/act2'
       */
      rtb_Switch_j = 0.0F;
    } else {
      rtb_Switch_j = CPP_Int_B->BusInput2.rPI_Dur_IntLimLo;
    }

    /* End of Switch: '<S31>/Switch2' */

    /* RelationalOperator: '<S34>/Limit Reached' */
    rtb_LimitReached = (CPP_Int_B->Saturadition >= rtb_Switch_j);

    /* Switch: '<S35>/Switch2' incorporates:
     *  Constant: '<S23>/act3'
     *  RelationalOperator: '<S35>/LowerRelop1'
     *  RelationalOperator: '<S35>/UpperRelop'
     *  Switch: '<S35>/Switch'
     */
    if (CPP_Int_B->BusInput2.rPI_Dur_IntLimHi > 1.0F) {
      rtb_rPr_AbsLimHi_k = 1.0F;
    } else if (CPP_Int_B->BusInput2.rPI_Dur_IntLimHi <
               CPP_Int_B->BusInput2.rPI_Dur_IntLimLo) {
      /* Switch: '<S35>/Switch' */
      rtb_rPr_AbsLimHi_k = CPP_Int_B->BusInput2.rPI_Dur_IntLimLo;
    } else {
      rtb_rPr_AbsLimHi_k = CPP_Int_B->BusInput2.rPI_Dur_IntLimHi;
    }

    /* End of Switch: '<S35>/Switch2' */

    /* Sum: '<S23>/Delta X' */
    rtb_rPr_AbsLim_h = rtb_rPr_AbsLimHi_k - rtb_Switch_j;

    /* Switch: '<S36>/Switch' incorporates:
     *  Abs: '<S36>/Abs'
     *  RelationalOperator: '<S36>/Relational Operator'
     */
    if (2.22044605E-16F >= (real32_T)fabs(rtb_rPr_AbsLim_h)) {
      rtb_rPr_AbsLim_h = 2.22044605E-16F;
    }

    /* End of Switch: '<S36>/Switch' */

    /* Product: '<S23>/y = k * (x - d)' incorporates:
     *  DataTypeConversion: '<S34>/Data Type Conversion'
     *  Gain: '<S8>/PI Duration reduction'
     *  Product: '<S32>/[k] - factor'
     *  Product: '<S34>/Enable Signal'
     *  Sum: '<S23>/Level Offset [x - d]'
     */
    rtb_Switch_j = ((real32_T)rtb_LimitReached * CPP_Int_B->Saturadition -
                    rtb_Switch_j) * (1.0F / rtb_rPr_AbsLim_h *
      -CPP_Int_B->BusInput1.rPI_Dur_Offset_Max);

    /* Switch: '<S33>/Switch2' incorporates:
     *  Constant: '<S23>/act1'
     *  Gain: '<S8>/PI Duration reduction'
     *  RelationalOperator: '<S33>/LowerRelop1'
     *  RelationalOperator: '<S33>/UpperRelop'
     *  Switch: '<S33>/Switch'
     */
    if (rtb_Switch_j > 0.0F) {
      rtb_Switch_j = 0.0F;
    } else {
      if (rtb_Switch_j < -CPP_Int_B->BusInput1.rPI_Dur_Offset_Max) {
        /* Switch: '<S33>/Switch' incorporates:
         *  Gain: '<S8>/PI Duration reduction'
         */
        rtb_Switch_j = -CPP_Int_B->BusInput1.rPI_Dur_Offset_Max;
      }
    }

    /* End of Switch: '<S33>/Switch2' */

    /* Product: '<S23>/Enable Output' incorporates:
     *  DataTypeConversion: '<S23>/Data Type Conversion'
     */
    CPP_Int_B->EnableOutput_m = (real32_T)rtb_LimitReached * rtb_Switch_j;
  }

  CPP_Int_PrevZCSigState->IgnitionPointandPIDurationOffse = (uint8_T)
    (rtb_LogicalOperator2 ? (int32_T)POS_ZCSIG : (int32_T)ZERO_ZCSIG);

  /* End of Outputs for SubSystem: '<Root>/Ignition Point and PI Duration Offset Calculator' */

  /* RelationalOperator: '<S39>/Compare' incorporates:
   *  Constant: '<S39>/Constant'
   */
  rtb_LogicalOperator2 = (CPP_Int_B->Saturadition >= 0.99F);

  /* RelationalOperator: '<S38>/Compare' incorporates:
   *  Constant: '<S38>/Constant'
   */
  rtb_LogicalOperator1_j = (CPP_Int_B->Saturadition > 0.0F);

  /* Logic: '<S10>/Sensor Error during Integrator Nonempty' */
  rtb_LimitReached = (CPP_Int_B->BusInput.bSensorErr && rtb_LogicalOperator1_j);

  /* Logic: '<S40>/Logical Operator2' */
  rtb_Reset = !rtb_LogicalOperator1_j;

  /* DiscreteIntegrator: '<S40>/Discrete-Time Accumulator' */
  if (rtb_Reset || (CPP_Int_DWork->DiscreteTimeAccumulator_PrevRes != 0)) {
    CPP_Int_DWork->DiscreteTimeAccumulator_DSTATE = 0.0F;
  }

  /* Logic: '<S40>/Logical Operator3' incorporates:
   *  DiscreteIntegrator: '<S40>/Discrete-Time Accumulator'
   *  RelationalOperator: '<S40>/Relational Operator'
   */
  rtb_LogicalOperator1_j = (rtb_LogicalOperator1_j &&
    (CPP_Int_DWork->DiscreteTimeAccumulator_DSTATE >=
     CPP_Int_B->BusInput2.tiInt_NonEmpty));

  /* Logic: '<S10>/Logical Operator3' */
  rtb_LimitReached = (rtb_LogicalOperator2 || rtb_LimitReached ||
                      rtb_LogicalOperator1_j);

  /* BusCreator: '<Root>/Bus Creator' incorporates:
   *  Logic: '<S10>/Logical Operator1'
   *  Logic: '<S10>/Logical Operator2'
   *  Logic: '<S10>/Logical Operator4'
   */
  CPP_Int_Y->tCPPI_OUT_c.rPr_CPP_Filt = CPP_Int_B->SensorErrorFilter;
  CPP_Int_Y->tCPPI_OUT_c.rPI_Dur_Offset = CPP_Int_B->EnableOutput_m;
  CPP_Int_Y->tCPPI_OUT_c.rCA_Ign_Offset = CPP_Int_B->EnableOutput;
  CPP_Int_Y->tCPPI_OUT_c.rNum_CPP_Int = CPP_Int_B->Saturadition;
  CPP_Int_Y->tCPPI_OUT_c.bCPP_AbsLim = ((!CPP_Int_B->BusInput.bLimpHomeExt) &&
    rtb_LimitReached);
  CPP_Int_Y->tCPPI_OUT_c.bCPP_AbsLim_LHE = (rtb_LimitReached &&
    CPP_Int_B->BusInput.bLimpHomeExt);
  CPP_Int_Y->tCPPI_OUT_c.bSkipCyl = rtb_LogicalOperator2;

  /* BusCreator: '<Root>/Bus Creator1' incorporates:
   *  DiscreteIntegrator: '<S40>/Discrete-Time Accumulator'
   */
  CPP_Int_Y->tCPPI_DBUG_o.tiInt_NonEmpty =
    CPP_Int_DWork->DiscreteTimeAccumulator_DSTATE;
  CPP_Int_Y->tCPPI_DBUG_o.rCPP_Err = CPP_Int_B->Divide3;
  CPP_Int_Y->tCPPI_DBUG_o.bECPG = rtb_FixPtRelationalOperator_h;
  CPP_Int_Y->tCPPI_DBUG_o.bFCPG = rtb_RelationalOperator1;

  /* S-Function (bur_bus_out): '<Root>/Bus Output' */
  inst->Out = CPP_Int_Y->tCPPI_OUT_c;

  /* S-Function (bur_bus_out): '<Root>/Bus Output1' */
  inst->Dbg = CPP_Int_Y->tCPPI_DBUG_o;

  /* Logic: '<S40>/Logical Operator1' */
  rtb_LogicalOperator1_j = !rtb_LogicalOperator1_j;

  /* Product: '<S40>/Block Windup' incorporates:
   *  DataTypeConversion: '<S40>/Data Type Conversion'
   */
  rtb_Switch_j = CPP_Int_B->BusInput.tiSample * (real32_T)rtb_LogicalOperator1_j;

  /* UnitDelay: '<S9>/Unit Delay' */
  CPP_Int_B->UnitDelay = CPP_Int_DWork->UnitDelay_DSTATE;

  /* S-Function (bur_out): '<Root>/Output3' */
  inst->Version = CPP_Int_B->UnitDelay;

  /* Update for UnitDelay: '<S1>/Unit Delay2' */
  CPP_Int_DWork->UnitDelay2_DSTATE = rtb_RelationalOperator1;

  /* Update for UnitDelay: '<S1>/Unit Delay1' */
  CPP_Int_DWork->UnitDelay1_DSTATE = rtb_FixPtRelationalOperator_h;

  /* Update for Delay: '<S1>/Engine Cycle Counter' */
  CPP_Int_DWork->EngineCycleCounter_DSTATE = rtb_Subtract3_h;

  /* Update for UnitDelay: '<S13>/Delay Input1' */
  CPP_Int_DWork->DelayInput1_DSTATE = CPP_Int_B->BusInput.rPr_CPP;

  /* Update for UnitDelay: '<S11>/Delay Input1' */
  CPP_Int_DWork->DelayInput1_DSTATE_c = rtb_LogicalOperator3;

  /* Update for Delay: '<S1>/Filter Cycle Counter' */
  CPP_Int_DWork->FilterCycleCounter_DSTATE = rtb_Subtract1;

  /* Update for UnitDelay: '<S4>/Delay Input1' */
  CPP_Int_DWork->DelayInput1_DSTATE_f = CPP_Int_B->BusInput.bReset;

  /* Update for DiscreteIntegrator: '<S40>/Discrete-Time Accumulator' */
  CPP_Int_DWork->DiscreteTimeAccumulator_DSTATE += rtb_Switch_j;
  if (rtb_Reset) {
    CPP_Int_DWork->DiscreteTimeAccumulator_PrevRes = 1;
  } else {
    CPP_Int_DWork->DiscreteTimeAccumulator_PrevRes = 0;
  }

  /* End of Update for DiscreteIntegrator: '<S40>/Discrete-Time Accumulator' */

  /* Update for UnitDelay: '<S9>/Unit Delay' */
  CPP_Int_DWork->UnitDelay_DSTATE = 10U;
}

/* Model initialize function */
void CPP_Int_initialize(struct PrevZCSigStates_CPP_Int *CPP_Int_PrevZCSigState, struct fCPP_Int* inst)
{
  CPP_Int_PrevZCSigState->IgnitionPointandPIDurationOffse = POS_ZCSIG;
  CPP_Int_PrevZCSigState->CylinderPeakPressureIntegrator_ = POS_ZCSIG;
  CPP_Int_PrevZCSigState->ResettableDelay_Reset_ZCE = UNINITIALIZED_ZCSIG;
  CPP_Int_PrevZCSigState->CylinderPeakPressureErrorCalcul = POS_ZCSIG;
}

/* Model terminate function */
void CPP_Int_terminate(struct fCPP_Int* inst)
{
  /* (no terminate code required) */
}

/*======================== TOOL VERSION INFORMATION ==========================*
 * MATLAB 8.0 (R2012b)20-Jul-2012                                             *
 * Simulink 8.0 (R2012b)20-Jul-2012                                           *
 * Simulink Coder 8.3 (R2012b)20-Jul-2012                                     *
 * Embedded Coder 6.3 (R2012b)20-Jul-2012                                     *
 *============================================================================*/

/*======================= LICENSE IN USE INFORMATION =========================*
 * matlab                                                                     *
 * matlab_coder                                                               *
 * real-time_workshop                                                         *
 * rtw_embedded_coder                                                         *
 * simulink                                                                   *
 *============================================================================*/
```

#### fCPP_Int.c
```c
/********************************************************************
 * COPYRIGHT -- Bernecker + Rainer Industrie-Elektronik Ges.m.b.H.
 ********************************************************************
 * Program: CPP_Int
 * File: fCPP_Int.c
 * Author: Messner
 * Created: Fri Nov 24 07:48:45 2017
 ********************************************************************
 * Implementation of program CPP_Int
 ********************************************************************
 * Generated with B&R Automation Studio Target for Simulink V4.2
 * (ERT based)
 ********************************************************************/
#include <bur/plctypes.h>
#include "CPP_Int.h"
#include "rtwtypes.h"

/* Defines */
#define SS_TERMINATE 4
#define SS_OUTPUT 3
#define SS_INITIALIZE 2

/*  Data Types */

/**************************** GLOBAL DATA *************************************/
/*  Definitions */

/*  Declarations  */

/***************************** FILE SCOPE DATA ********************************/

/*************************** FUNCTIONS ****************************************/
#ifdef __cplusplus

unsigned long bur_heap_size = 6553500;

#endif

void fCPP_Int(struct fCPP_Int* inst)
{
  BlockIO_CPP_Int *CPP_Int_B = &(inst)->bur_BlockIO_CPP_Int;
	D_Work_CPP_Int *CPP_Int_DWork = &(inst)->bur_D_Work_CPP_Int;
	PrevZCSigStates_CPP_Int *CPP_Int_PrevZCSigState = &(inst)->bur_PrevZCSigStates_CPP_Int;
	ExternalOutputs_CPP_Int *CPP_Int_Y = &(inst)->bur_ExternalOutputs_CPP_Int;

  switch (inst->ssMethodType)
  {
   case SS_INITIALIZE:
    /* call model initialize function */
    CPP_Int_initialize(CPP_Int_PrevZCSigState, inst);
    break;

   case SS_OUTPUT:
    /* call model step function */
    CPP_Int_step(CPP_Int_B, CPP_Int_DWork, CPP_Int_PrevZCSigState, CPP_Int_Y, inst);

    break;

   case SS_TERMINATE:
    /* call model terminate function */
    CPP_Int_terminate(inst);
    break;
  }
}

/*****************************************************************************
   Function block sample time: 0.01s
 *****************************************************************************/

/*****************************************************************************
   B&R Automation Studio Target for Simulink Version: A4.5.1 (27-Jul-2015)
 *****************************************************************************/

/*======================== TOOL VERSION INFORMATION ==========================*
 * MATLAB 8.0 (R2012b)20-Jul-2012                                             *
 * Simulink 8.0 (R2012b)20-Jul-2012                                           *
 * Simulink Coder 8.3 (R2012b)20-Jul-2012                                     *
 * Embedded Coder 6.3 (R2012b)20-Jul-2012                                     *
 *============================================================================*/

/*======================= LICENSE IN USE INFORMATION =========================*
 * matlab                                                                     *
 * matlab_coder                                                               *
 * real-time_workshop                                                         *
 * rtw_embedded_coder                                                         *
 * simulink                                                                   *
 *============================================================================*/
```

#### lib_properties.txt
```
For manual assignment to hardware configuration please
add the following additional include directories:

\Logical\MATLAB_includes\R2012b\

And the following additional build options:

-lm -D MODEL=CPP_Int -D NUMST=1 -D NCSTATES=0 -D HAVESTDIO -D ONESTEPFCN=1 -D TERMFCN=1 -D MAT_FILE=0 -D MULTI_INSTANCE_CODE=1 -D INTEGER_CODE=0 -D MT=0 -D CLASSIC_INTERFACE=0 -D TID01EQ=0
```

### Library Logical/EngineController/Lib_EC/lLX2 (ANSIC)

#### lLX2.fun
```iecst
FUNCTION_BLOCK fLX2
  VAR_INPUT
    ssMethodType: SINT;
  END_VAR  VAR_INPUT
        IN : tLX2_IN; (**)
  END_VAR
  VAR_INPUT
        PERM : tLX2_PERM; (**)
  END_VAR
  VAR_INPUT
        PARA : tLX2_PARA; (**)
  END_VAR
 VAR_OUTPUT
        Output : tLX2_OUT; (**)
  END_VAR
 VAR_OUTPUT
        DBUG : tLX2_DBUG; (**)
  END_VAR
  VAR_OUTPUT
        Version : UDINT; (**)
  END_VAR
	VAR
		bur_BlockIO_LX2 : BlockIO_LX2;
	END_VAR
	VAR
		bur_D_Work_LX2 : D_Work_LX2;
	END_VAR
	VAR
		bur_ExternalInputs_LX2 : ExternalInputs_LX2;
	END_VAR
	VAR
		bur_ExternalOutputs_LX2 : ExternalOutputs_LX2;
	END_VAR
	VAR
		bur_LX2 : tag_RTM_LX2;
	END_VAR
END_FUNCTION_BLOCK
```

#### lLX2.typ
```iecst
TYPE

   tLX2_CTR_DBUG : STRUCT
        rCtrlError : REAL; (*Error between NOx,set and NOx,act_filt [ppm]*)
        rPr_offset_Ctrl : REAL; (*Output of I-Controler [bar]*)
        rPr_LX2_offset_preSat : REAL; (*LX2 delta_p2s_LX2 before Saturation [bar]*)
        bLX2_inSaturation : BOOL; (*true, if LX2 is in Saturation*)
        rNOx_act_filt : REAL; (*filtered NOx signal [ppm]*)
        rPr_Ctrl_LowerLim_act : REAL; (*Controler Output - Lower Limit actuel [bar]*)
        rPr_Ctrl_UpperLim_act : REAL; (*Controler Output - Upper Limit actuel [bar]*)
        rPr_offset_BPOC_all : REAL; (*interpolated delta_p2s from BPOC_Gas 1-4 [bar]*)
        rPr_y0_Ctrl : REAL; (*initial conditions of controler [bar]*)
        rLX2_inLimit_Timer : REAL; (*Timer, LX2 in Limit [sec]*)
        bLX2_inLimit_NoDelay : BOOL; (*true, if LX2 control limit is reached*)
    END_STRUCT;

   tLX2_DBUG : STRUCT
        Stm : tLX2_STM_DBUG; (*debugging state machine*)
        Ctr : tLX2_CTR_DBUG; (*debugging controller*)
        Gas1 : tLX2_GAS_DBUG; (*debugging BPOC Gas 1*)
        Gas2 : tLX2_GAS_DBUG; (*debugging BPOC Gas 2*)
        Gas3 : tLX2_GAS_DBUG; (*debugging BPOC Gas 3*)
        Gas4 : tLX2_GAS_DBUG; (*debugging BPOC Gas 4*)
        rLX2_BPOC_internal : ARRAY[0..10] OF REAL; (*LX2 BPOC - delta p2s at all node points - internal [bar]*)
        bLX2_BPOC_measured_internal : ARRAY[0..10] OF BOOL; (*LX2 BPOC - binary map of already measured points - internal [true->measured]*)
        rBPOC_Lp_all : ARRAY[0..2] OF REAL; (*position of Leanox points (b,a,c) at BPOC_all [0...1]*)
    END_STRUCT;

   tLX2_GAS_DBUG : STRUCT
        bBPOC_enable : BOOL; (*true, if BPOC is used to generate delta_p2s*)
        bBPOC_save_enable : BOOL; (*BPOC will be updated, [true->learning=on]*)
        bBPOC_measured_map_IN : ARRAY[0..10] OF BOOL; (*Input of BPOC manipulation algorithm, measered nodes [bool]*)
        rBPOC_offset_map_IN : ARRAY[0..10] OF REAL; (*Input of BPOC manipulation algorithm, p2s offsets [bar]*)
        rPr_BPOC_offset_IN : REAL; (*Input of BPOC manipulation algorithm, desired p2s_offsets [bar]*)
        bBPOC_measured_map_OUT : ARRAY[0..10] OF BOOL; (*Output of BPOC_Gas manipulation algorithm, measered nodes [bool]*)
        rBPOC_offset_map_OUT : ARRAY[0..10] OF REAL; (*Output of BPOC manipulation algorithm, p2s offsets [bar]*)
        rPr_BPOC_offset_OUT : REAL; (*Output, interpolated delta_p2s from BPOC [bar]*)
        rP_act_Norm_Filt : REAL; (*Power setpoint related to rP_Nom [0...1]*)
        rLX2_BPOC_Error : REAL; (*Error between BPOC and new p2s [bar]*)
        rLX2_Lp : ARRAY[0..2] OF REAL; (*position of Leanox Points (b,a,c) [%-EngPower]*)
        rBPOC_DBUG_a : ARRAY[0..1] OF REAL; (*weighting factors due to leverage function [0...1]*)
        rBPOC_DBUG_b : ARRAY[0..1] OF REAL; (*indices of affected node points due to new measurement value [1...11]*)
        rBPOC_DBUG_Lp : ARRAY[0..3] OF REAL; (*position of Leanox points (0kW,b,a,c) at BPOC [0...1]*)
        rBPOC_DBUG_s : ARRAY[0..2] OF REAL; (*calculated slope between two affected nodes due to leverage function; Gas [0...1]*)
    END_STRUCT;

   tLX2_IN : STRUCT
        bLX2_active : BOOL; (*LX2 active*)
        rNOx_act : REAL; (*Actual NOx value [ppm]*)
        rNOx_set : REAL; (*NOx reference value [ppm]*)
        bNOx_valid : BOOL; (*NOx signal valid*)
        rP_Set_Norm : REAL; (*Power setpoint related to rP_Nom [0...1]*)
        rP_Lp_b : ARRAY[0..4] OF REAL; (*P at Leanox point b (half Load) - Gas 1/2/3/4 [kW]*)
        rP_Lp_a : ARRAY[0..4] OF REAL; (*P at Leanox point a (full Load) - Gas 1/2/3/4[kW]*)
        rP_Lp_c : ARRAY[0..4] OF REAL; (*P at Leanox point c (~25% Load) - Gas 1/2/3/4 [kW]*)
        bLp_c_ena : BOOL; (*Leanox point c enabled [true->enabled]*)
        rP_Nom : ARRAY[0..4] OF REAL; (*Engine Power Output Nominell - Gas 1/2/3/4 [kW]*)
        bESC_active : BOOL; (*ESC control active [true->ESC on]*)
        bBPOC_reset : BOOL; (*Reset BPOC [true->for one cycle]*)
        bLeanox_Engine_Man : BOOL; (*Leanox mode [true->manual]*)
        bLeanox_Adjust : BOOL; (*Leanox save - confirm button [true->for one cycle]*)
        rKnock_level : REAL; (*max. Knockintegrator value of all Zylinder [0...1]*)
        rMisfire_level : REAL; (*misfire integrator value - detection via power fluctuation [0...1]*)
        rGT_QualMix_1_2 : REAL; (*gas mixing ratio Gas1/Gas2 [0...1] (0=>100% Gas 1)*)
        rGT_RatioMix : REAL; (*gas mixing ratio Gas0/Gas3 [0...1] (0=>100% Gas 0)*)
        iIdx_Gtyp_Dem : UINT; (*Gastype [0...4] (0=Gasmixing, 1=Gas 1, 2=Gas 2, 3=Gas 3, 4=Gas 4)*)
        rLX2_BPOC_Gas1 : ARRAY[0..10] OF REAL; (*actual BPOC from Permanent Storage - Gas 1 [bar]*)
        bLX2_BPOC_measured_Gas1 : ARRAY[0..10] OF BOOL; (*LX2 BPOC - binary map of already measured points - Gas 1 [true->measured]*)
        rLX2_BPOC_Gas2 : ARRAY[0..10] OF REAL; (*actual BPOC from Permanent Storage - Gas 1 [bar]*)
        bLX2_BPOC_measured_Gas2 : ARRAY[0..10] OF BOOL; (*LX2 BPOC - binary map of already measured points - Gas 2 [true->measured]*)
        rLX2_BPOC_Gas3 : ARRAY[0..10] OF REAL; (*actual BPOC from Permanent Storage - Gas 2 [bar]*)
        bLX2_BPOC_measured_Gas3 : ARRAY[0..10] OF BOOL; (*LX2 BPOC - binary map of already measured points - Gas 3 [true->measured]*)
        rLX2_BPOC_Gas4 : ARRAY[0..10] OF REAL; (*actual BPOC from Permanent Storage - Gas 3 [bar]*)
        bLX2_BPOC_measured_Gas4 : ARRAY[0..10] OF BOOL; (*LX2 BPOC - binary map of already measured points - Gas 4 [true->measured]*)
        rPr_Leanox_Dev : REAL; (*Leanox controller deviation [mbar]*)
        bExt_SteadyState_Loss : BOOL; (*External interface signal for steady state loss [true->no steady state]*)
        bExt_BPOC_learning_Stop : BOOL; (*External interface signal for BPOC learning stop [true->no BPOC learning]*)
        bLX2_fastRamp : BOOL; (*Fast ramp request [true->fast ramp on]*)
        rLX2_fastRampMult : REAL; (*Fast ramp multiplier, applied to default rate limit if requested*)
    END_STRUCT;

   tLX2_OUT : STRUCT
        rPr_LX2_offset : REAL; (*LX2 boost pressure offset - delta p2s_LX2 [bar]*)
        bLX2_save : ARRAY[0..4] OF BOOL; (*save LX2 data, Gas 1-4, [true->save]*)
        rPr_LX2_offset_Lp_b : ARRAY[0..4] OF REAL; (*LX2 - delta p2s at Leanox point b (half load), Gas 1-4, [bar]*)
        rPr_LX2_offset_Lp_a : ARRAY[0..4] OF REAL; (*LX2 - delta p2s at Leanox point a (full load), Gas 1-4,  [bar]*)
        rPr_LX2_offset_Lp_c : ARRAY[0..4] OF REAL; (*LX2 - delta p2s at Leanox point c (~25% load), Gas 1-4,  [bar]*)
        rLX2_BPOC_Gas1 : ARRAY[0..10] OF REAL; (*LX2 BPOC - delta p2s at all node points - Gas 1[bar]*)
        bLX2_BPOC_measured_Gas1 : ARRAY[0..10] OF BOOL; (*LX2 BPOC - binary map of already measured points - Gas 1 [true->measured]*)
        rLX2_BPOC_Gas2 : ARRAY[0..10] OF REAL; (*LX2 BPOC - delta p2s at all node points - Gas 2 [bar]*)
        bLX2_BPOC_measured_Gas2 : ARRAY[0..10] OF BOOL; (*LX2 BPOC - binary map of already measured points - Gas 2 [true->measured]*)
        rLX2_BPOC_Gas3 : ARRAY[0..10] OF REAL; (*LX2 BPOC - delta p2s at all node points - Gas 3 [bar]*)
        bLX2_BPOC_measured_Gas3 : ARRAY[0..10] OF BOOL; (*LX2 BPOC - binary map of already measured points - Gas 3 [true->measured]*)
        rLX2_BPOC_Gas4 : ARRAY[0..10] OF REAL; (*LX2 BPOC - delta p2s at all node points - Gas 4 [bar]*)
        bLX2_BPOC_measured_Gas4 : ARRAY[0..10] OF BOOL; (*LX2 BPOC - binary map of already measured points - Gas 4 [true->measured]*)
        rLX2_BPOC : ARRAY[0..10] OF REAL; (*LX2 BPOC,act (all Gases combined) - delta p2s at all node points [bar]*)
        bLX2_BPOC_measured : ARRAY[0..10] OF BOOL; (*LX2 BPOC,measured (all Gases combined) - binary map of already measured points [true->measured]*)
        bBPOC_enable : BOOL; (*FOR VISU: true, if one out of 4 BPOCs is used to generate delta_p2s, Gas 1-4, [0/1]*)
        bBPOC_save_enable : BOOL; (*FOR VISU: if true; one out of 4 BPOCs will be updated, [true->learning=on], Gas 1-4, [0/1]*)
        bLX2_inLimit : BOOL; (*FOR Warning: if true; LX2 is in Limit and Warning shall appear[true->in Limit], [0/1]*)
    END_STRUCT;

   tLX2_PARA : STRUCT
        bLX2_enable : BOOL; (*enable LX2*)
        rLX2_Ctrl_Tn : REAL; (*Ctrl Integrator time constant [sec]*)
        rFilterConst_NOx : REAL; (*Filter coefficient PT1 - NOx act [sec]*)
        rPr_LX2_OffsetLimit : REAL; (*LX2 charge pressure offset limit [mbar]*)
        rLX2_SteadyStateFactor : REAL; (*Steady state factor for LX2*)
    END_STRUCT;

   tLX2_PERM : STRUCT
        iWeight_Lp_0kW : UINT; (*weighting of Leanox point 0kW [0..65535]*)
        iWeight_Lp_b : UINT; (*weighting of Leanox point b (half load), UserDefine [0..65535]*)
        iWeight_Lp_a : UINT; (*weighting of Leanox point a (full load) [0..65535]*)
        iWeight_Lp_c : UINT; (*weighting of Leanox point c (~25% load) [0..65535]*)
        rThreshold_knock : REAL; (*Knocking Threshold - LX2 knows about knocking [0...1]*)
        rThreshold_misfire : REAL; (*Misfire Threshold - LX2 knows about misfire [0...1]*)
        iCtrl_RateLimit_TraceBack : UINT; (*Rate limit for tracing Controler back to zero; mbar/sec [0..65535]*)
        iFilterConst_P_set : UINT; (*Filter coefficient PT1 - P_set [sec]*)
        rThreshold_save2map : ARRAY[0..1] OF REAL; (*Threshold at which amount of gas the map will be updated [0...1]*)
        rLX2_inLimitSetup_Time : REAL; (*tolerated rTime_inSaturation [0...x sec]*)
        iTiUpdate_BPOC : UINT; (*Update Time of BPOC [sec]*)
        iTiDelay_SteadyState : UINT; (*Delay timer for LX2 steady state [sec]*)
        iFiltConst_LeanoxDev_SteadyState : UINT; (*Filter coefficient PT1 - Leanox deviation for LX2 steady state [sec]*)
        iFiltConst_P_set_SteadyState : UINT; (*Filter coefficient PT1 - norm. power setpoint for LX2 steady state [sec]*)
        rThreshold_LeanoxDev_SteadyState : REAL; (*Threshold leanox deviation for LX2 steady state [mbar]*)
        rThreshold_P_set_SteadyState : REAL; (*Threshold norm. power setpoint steady for LX2 steady state [0...1]*)
        rCtrlError_Limit : REAL; (*Saturation limit for error between NOx_set and NOx_act_filt [ppm]*)
    END_STRUCT;

   tLX2_STM_DBUG : STRUCT
        rP_act_Norm_Filt : REAL; (*Power setpoint filtered related to rP_Nom [0...100]*)
        bBPOC_enable : ARRAY[0..3] OF BOOL; (*true, if BPOC is used to generate delta_p2s, Gas 1-4, [0/1]*)
        bBPOC_save_enable : ARRAY[0..3] OF BOOL; (*if true; BPOC will be updated, [true->learning=on], Gas 1-4, [0/1]*)
        rSplitfactor_Gas : ARRAY[0..3] OF REAL; (*indicates how much of each gas is taking part on combustion, Gas 1-4 [0...1]*)
        bCtrl_enable : BOOL; (*true, if Controler is enabled*)
        bCtrl_freeze : BOOL; (*true, if Controler is frozen*)
        bEng_knock : BOOL; (*true, if engine is knocking due to LX2 rules*)
        bEng_misfire : BOOL; (*true, if engine is misfiring due to LX2 rules*)
        bBPOC_reset : BOOL; (*if true; BPOC will be reset, [0/1]*)
        iTimer_save : UINT; (*Timer of Save Logic [sec]*)
        bLX2_SteadyState : BOOL; (*true, if engine in steady state operation as per LX2 definition*)
        bLX2_SteadyState_noDelay : BOOL; (*true, if engine in steady state operation as per LX2 definition without delay timer*)
        bLX2_LeanoxDev_Steady : BOOL; (*true, if leanox deviation within limit as per LX2 steady state definition*)
        bLX2_P_Set_Steady : BOOL; (*true, if power setpoint steady as per LX2 steady state definition*)
    END_STRUCT;
END_TYPE
TYPE
rtB_BoostPressureOffsetCurve_LX : STRUCT
	OUT_offset : ARRAY[0..10] OF REAL;
	e : REAL;
	DBUG_a : ARRAY[0..1] OF REAL;
	DBUG_b : ARRAY[0..1] OF REAL;
	DBUG_Lp : ARRAY[0..3] OF REAL;
	DBUG_s : ARRAY[0..2] OF REAL;
	OUT_measured : ARRAY[0..10] OF BOOL;
END_STRUCT;
rtB_TON_LX2 : STRUCT
	DiscreteTimeIntegrator : REAL;
	LogicalOperator3 : BOOL;
END_STRUCT;
rtDW_TON_LX2 : STRUCT
	DiscreteTimeIntegrator_DSTATE : REAL;
	DiscreteTimeIntegrator_PrevRese : SINT;
END_STRUCT;
rtB_Filter1_LX2 : STRUCT
	Switch : REAL;
END_STRUCT;
rtDW_Filter1_LX2 : STRUCT
	DiscreteTimeIntegrator_DSTATE : REAL;
	DiscreteTimeIntegrator_PrevRese : SINT;
	DiscreteTimeIntegrator_IC_LOADI : USINT;
END_STRUCT;
BlockIO_LX2 : STRUCT
	BusInput : tLX2_IN;
	BusInput1 : tLX2_PERM;
	BusInput2 : tLX2_PARA;
	UnitDelay : UDINT;
	TON_p : rtB_TON_LX2;
	Filter1 : rtB_Filter1_LX2;
	Filter : rtB_Filter1_LX2;
	Filter1_i : rtB_Filter1_LX2;
	TON_b : rtB_TON_LX2;
	sf_BoostPressureOffsetCurve_a : rtB_BoostPressureOffsetCurve_LX;
	sf_BoostPressureOffsetCurve_d : rtB_BoostPressureOffsetCurve_LX;
	sf_BoostPressureOffsetCurve_f : rtB_BoostPressureOffsetCurve_LX;
	sf_BoostPressureOffsetCurve : rtB_BoostPressureOffsetCurve_LX;
END_STRUCT;
D_Work_LX2 : STRUCT
	UnitDelay3_DSTATE : REAL;
	Delay2_DSTATE : ARRAY[0..10] OF REAL;
	UnitDelay2_DSTATE : REAL;
	Delay2_DSTATE_j : ARRAY[0..10] OF REAL;
	Delay2_DSTATE_b : ARRAY[0..10] OF REAL;
	Delay2_DSTATE_d : ARRAY[0..10] OF REAL;
	UnitDelay5_DSTATE : REAL;
	UnitDelay6_DSTATE : REAL;
	DiscreteTimeIntegrator_DSTATE : REAL;
	UnitDelay4_DSTATE : REAL;
	Delay_DSTATE : REAL;
	DiscreteTimeIntegrator_DSTATE_n : REAL;
	UnitDelay_DSTATE : UDINT;
	y0_1 : REAL;
	DiscreteTimeIntegrator_DSTATE_l : UINT;
	UnitDelay1_DSTATE : BOOL;
	UnitDelay1_DSTATE_l : BOOL;
	UnitDelay_DSTATE_l : BOOL;
	Delay1_DSTATE : ARRAY[0..10] OF BOOL;
	Delay1_DSTATE_l : ARRAY[0..10] OF BOOL;
	Delay1_DSTATE_o : ARRAY[0..10] OF BOOL;
	Delay1_DSTATE_g : ARRAY[0..10] OF BOOL;
	DelayInput1_DSTATE : BOOL;
	DiscreteTimeIntegrator_PrevRese : SINT;
	DiscreteTimeIntegrator_PrevRe_m : SINT;
	DiscreteTimeIntegrator_PrevRe_a : SINT;
	icLoad : USINT;
	icLoad_o : USINT;
	icLoad_or : USINT;
	icLoad_oj : USINT;
	icLoad_p : USINT;
	icLoad_d : USINT;
	icLoad_f : USINT;
	icLoad_c : USINT;
	DiscreteTimeIntegrator_IC_LOADI : USINT;
	icLoad_i : USINT;
	DiscreteTimeIntegrator_IC_LOA_l : USINT;
	TON_p : rtDW_TON_LX2;
	Filter1 : rtDW_Filter1_LX2;
	Filter : rtDW_Filter1_LX2;
	Filter1_i : rtDW_Filter1_LX2;
	TON_b : rtDW_TON_LX2;
END_STRUCT;
PrevZCSigStates_LX2 : STRUCT
	Delay2_Reset_ZCE : USINT;
	Delay1_Reset_ZCE : USINT;
	Delay2_Reset_ZCE_o : USINT;
	Delay1_Reset_ZCE_n : USINT;
	Delay2_Reset_ZCE_or : USINT;
	Delay1_Reset_ZCE_e : USINT;
	Delay2_Reset_ZCE_k : USINT;
	Delay1_Reset_ZCE_k : USINT;
	Delay_Reset_ZCE : USINT;
END_STRUCT;
ConstParam_LX2 : STRUCT
	pooled14 : ARRAY[0..10] OF REAL;
END_STRUCT;
ExternalInputs_LX2 : STRUCT
	tLX2_IN_e : tLX2_IN;
	tLX2_PERM_m : tLX2_PERM;
	tLX2_PARA_c : tLX2_PARA;
END_STRUCT;
ExternalOutputs_LX2 : STRUCT
	tLX2_OUT_c : tLX2_OUT;
	tLX2_DBUG_j : tLX2_DBUG;
END_STRUCT;
tag_RTM_LX2 : STRUCT
	errorStatus : REFERENCE TO USINT;
END_STRUCT;
END_TYPE
```
